   1:  PR[GP1:91,1] = PR[GP1:90,1] + 45.256;
   1:  PR[GP1:91,2] = PR[GP1:90,2] + 33.869;
   1:L PR[91] 10mm/sec CNT100;
   1:  PR[GP1:91,1] = PR[GP1:90,1] + 42.073;
   1:  PR[GP1:91,2] = PR[GP1:90,2] + 34.713;
   1:L PR[91] 10mm/sec CNT100;
   1:  PR[GP1:91,1] = PR[GP1:90,1] + 30.579;
   1:  PR[GP1:91,2] = PR[GP1:90,2] + 34.067;
   1:L PR[91] 10mm/sec CNT100;
   1:  PR[GP1:91,1] = PR[GP1:90,1] + 29.717;
   1:  PR[GP1:91,2] = PR[GP1:90,2] + 33.970;
   1:L PR[91] 10mm/sec CNT100;
   1:  PR[GP1:91,1] = PR[GP1:90,1] + 25.402;
   1:  PR[GP1:91,2] = PR[GP1:90,2] + 32.076;
   1:L PR[91] 10mm/sec CNT100;
   1:  PR[GP1:91,1] = PR[GP1:90,1] + 18.379;
   1:  PR[GP1:91,2] = PR[GP1:90,2] + 29.146;
   1:L PR[91] 10mm/sec CNT100;
   1:  PR[GP1:91,1] = PR[GP1:90,1] + 17.053;
   1:  PR[GP1:91,2] = PR[GP1:90,2] + 28.085;
   1:L PR[91] 10mm/sec CNT100;
   1:  PR[GP1:91,1] = PR[GP1:90,1] + 9.465;
   1:  PR[GP1:91,2] = PR[GP1:90,2] + 20.933;
   1:L PR[91] 10mm/sec CNT100;
   1:  PR[GP1:91,1] = PR[GP1:90,1] + 7.394;
   1:  PR[GP1:91,2] = PR[GP1:90,2] + 17.518;
   1:L PR[91] 10mm/sec CNT100;
   1:  PR[GP1:91,1] = PR[GP1:90,1] + 3.717;
   1:  PR[GP1:91,2] = PR[GP1:90,2] + 9.866;
   1:L PR[91] 10mm/sec CNT100;
   1:  PR[GP1:91,1] = PR[GP1:90,1] + -4.263;
   1:L PR[91] 10mm/sec CNT100;
   1:  PR[GP1:91,1] = PR[GP1:90,1] + -7.931;
   1:  PR[GP1:91,2] = PR[GP1:90,2] + 17.537;
   1:L PR[91] 10mm/sec CNT100;
   1:  PR[GP1:91,1] = PR[GP1:90,1] + -10.000;
   1:  PR[GP1:91,2] = PR[GP1:90,2] + 20.955;
   1:L PR[91] 10mm/sec CNT100;
   1:  PR[GP1:91,1] = PR[GP1:90,1] + -17.593;
   1:  PR[GP1:91,2] = PR[GP1:90,2] + 28.093;
   1:L PR[91] 10mm/sec CNT100;
   1:  PR[GP1:91,1] = PR[GP1:90,1] + -18.917;
   1:  PR[GP1:91,2] = PR[GP1:90,2] + 29.150;
   1:L PR[91] 10mm/sec CNT100;
   1:  PR[GP1:91,1] = PR[GP1:90,1] + -25.929;
   1:  PR[GP1:91,2] = PR[GP1:90,2] + 32.075;
   1:L PR[91] 10mm/sec CNT100;
   1:  PR[GP1:91,1] = PR[GP1:90,1] + -30.255;
   1:  PR[GP1:91,2] = PR[GP1:90,2] + 33.974;
   1:L PR[91] 10mm/sec CNT100;
   1:  PR[GP1:91,1] = PR[GP1:90,1] + -31.120;
   1:  PR[GP1:91,2] = PR[GP1:90,2] + 34.071;
   1:L PR[91] 10mm/sec CNT100;
   1:  PR[GP1:91,1] = PR[GP1:90,1] + -42.608;
   1:  PR[GP1:91,2] = PR[GP1:90,2] + 34.711;
   1:L PR[91] 10mm/sec CNT100;
   1:  PR[GP1:91,1] = PR[GP1:90,1] + -45.793;
   1:  PR[GP1:91,2] = PR[GP1:90,2] + 33.866;
   1:L PR[91] 10mm/sec CNT100;
   1:  PR[GP1:91,1] = PR[GP1:90,1] + -54.608;
   1:  PR[GP1:91,2] = PR[GP1:90,2] + 31.119;
   1:L PR[91] 10mm/sec CNT100;
   1:  PR[GP1:91,1] = PR[GP1:90,1] + -58.773;
   1:  PR[GP1:91,2] = PR[GP1:90,2] + 28.074;
   1:L PR[91] 10mm/sec CNT100;
   1:  PR[GP1:91,1] = PR[GP1:90,1] + -64.659;
   1:  PR[GP1:91,2] = PR[GP1:90,2] + 23.496;
   1:L PR[91] 10mm/sec CNT100;
   1:  PR[GP1:91,1] = PR[GP1:90,1] + -68.074;
   1:  PR[GP1:91,2] = PR[GP1:90,2] + 18.107;
   1:L PR[91] 10mm/sec CNT100;
   1:  PR[GP1:91,1] = PR[GP1:90,1] + -71.344;
   1:  PR[GP1:91,2] = PR[GP1:90,2] + 12.729;
   1:L PR[91] 10mm/sec CNT100;
   1:  PR[GP1:91,1] = PR[GP1:90,1] + -72.694;
   1:  PR[GP1:91,2] = PR[GP1:90,2] + 5.689;
   1:L PR[91] 10mm/sec CNT100;
   1:  PR[GP1:91,1] = PR[GP1:90,1] + -73.693;
   1:  PR[GP1:91,2] = PR[GP1:90,2] + 0.281;
   1:L PR[91] 10mm/sec CNT100;
   1:  PR[GP1:91,1] = PR[GP1:90,1] + -72.360;
   1:  PR[GP1:91,2] = PR[GP1:90,2] + -6.656;
   1:L PR[91] 10mm/sec CNT100;
   1:  PR[GP1:91,1] = PR[GP1:90,1] + -71.343;
   1:  PR[GP1:91,2] = PR[GP1:90,2] + -12.173;
   1:L PR[91] 10mm/sec CNT100;
   1:  PR[GP1:91,1] = PR[GP1:90,1] + -68.074;
   1:  PR[GP1:91,2] = PR[GP1:90,2] + -17.549;
   1:L PR[91] 10mm/sec CNT100;
   1:  PR[GP1:91,1] = PR[GP1:90,1] + -64.659;
   1:  PR[GP1:91,2] = PR[GP1:90,2] + -22.938;
   1:L PR[91] 10mm/sec CNT100;
   1:  PR[GP1:91,1] = PR[GP1:90,1] + -58.773;
   1:  PR[GP1:91,2] = PR[GP1:90,2] + -27.516;
   1:L PR[91] 10mm/sec CNT100;
   1:  PR[GP1:91,1] = PR[GP1:90,1] + -54.608;
   1:  PR[GP1:91,2] = PR[GP1:90,2] + -30.561;
   1:L PR[91] 10mm/sec CNT100;
   1:  PR[GP1:91,1] = PR[GP1:90,1] + -45.793;
   1:  PR[GP1:91,2] = PR[GP1:90,2] + -33.308;
   1:L PR[91] 10mm/sec CNT100;
   1:  PR[GP1:91,1] = PR[GP1:90,1] + -42.608;
   1:  PR[GP1:91,2] = PR[GP1:90,2] + -34.153;
   1:L PR[91] 10mm/sec CNT100;
   1:  PR[GP1:91,1] = PR[GP1:90,1] + -31.120;
   1:  PR[GP1:91,2] = PR[GP1:90,2] + -33.513;
   1:L PR[91] 10mm/sec CNT100;
   1:  PR[GP1:91,1] = PR[GP1:90,1] + -30.255;
   1:  PR[GP1:91,2] = PR[GP1:90,2] + -33.416;
   1:L PR[91] 10mm/sec CNT100;
   1:  PR[GP1:91,1] = PR[GP1:90,1] + -25.929;
   1:  PR[GP1:91,2] = PR[GP1:90,2] + -31.517;
   1:L PR[91] 10mm/sec CNT100;
   1:  PR[GP1:91,1] = PR[GP1:90,1] + -18.917;
   1:  PR[GP1:91,2] = PR[GP1:90,2] + -28.592;
   1:L PR[91] 10mm/sec CNT100;
   1:  PR[GP1:91,1] = PR[GP1:90,1] + -17.593;
   1:  PR[GP1:91,2] = PR[GP1:90,2] + -27.535;
   1:L PR[91] 10mm/sec CNT100;
   1:  PR[GP1:91,1] = PR[GP1:90,1] + -10.000;
   1:  PR[GP1:91,2] = PR[GP1:90,2] + -20.397;
   1:L PR[91] 10mm/sec CNT100;
   1:  PR[GP1:91,1] = PR[GP1:90,1] + -7.931;
   1:  PR[GP1:91,2] = PR[GP1:90,2] + -16.979;
   1:L PR[91] 10mm/sec CNT100;
   1:  PR[GP1:91,1] = PR[GP1:90,1] + -4.250;
   1:  PR[GP1:91,2] = PR[GP1:90,2] + -9.308;
   1:L PR[91] 10mm/sec CNT100;
   1:  PR[GP1:91,1] = PR[GP1:90,1] + 3.730;
   1:L PR[91] 10mm/sec CNT100;
   1:  PR[GP1:91,1] = PR[GP1:90,1] + 6.788;
   1:  PR[GP1:91,2] = PR[GP1:90,2] + -16.217;
   1:  PR[GP1:91,3] = PR[GP1:90,3] + 25.925;
   1:L PR[91] 10mm/sec CNT100;
   1:  PR[GP1:91,1] = PR[GP1:90,1] + 9.452;
   1:  PR[GP1:91,2] = PR[GP1:90,2] + -20.613;
   1:L PR[91] 10mm/sec CNT100;
   1:  PR[GP1:91,1] = PR[GP1:90,1] + 16.180;
   1:  PR[GP1:91,2] = PR[GP1:90,2] + -26.953;
   1:L PR[91] 10mm/sec CNT100;
   1:  PR[GP1:91,1] = PR[GP1:90,1] + 18.397;
   1:  PR[GP1:91,2] = PR[GP1:90,2] + -28.727;
   1:L PR[91] 10mm/sec CNT100;
   1:  PR[GP1:91,1] = PR[GP1:90,1] + 29.756;
   1:  PR[GP1:91,2] = PR[GP1:90,2] + -33.465;
   1:L PR[91] 10mm/sec CNT100;
   1:  PR[GP1:91,1] = PR[GP1:90,1] + 42.107;
   1:  PR[GP1:91,2] = PR[GP1:90,2] + -34.158;
   1:L PR[91] 10mm/sec CNT100;
   1:  PR[GP1:91,1] = PR[GP1:90,1] + 44.426;
   1:  PR[GP1:91,2] = PR[GP1:90,2] + -33.543;
   1:L PR[91] 10mm/sec CNT100;
   1:  PR[GP1:91,1] = PR[GP1:90,1] + 54.074;
   1:  PR[GP1:91,2] = PR[GP1:90,2] + -30.539;
   1:L PR[91] 10mm/sec CNT100;
   1:  PR[GP1:91,1] = PR[GP1:90,1] + 57.584;
   1:  PR[GP1:91,2] = PR[GP1:90,2] + -27.974;
   1:L PR[91] 10mm/sec CNT100;
   1:  PR[GP1:91,1] = PR[GP1:90,1] + 64.095;
   1:  PR[GP1:91,2] = PR[GP1:90,2] + -22.908;
   1:L PR[91] 10mm/sec CNT100;
   1:  PR[GP1:91,1] = PR[GP1:90,1] + 67.111;
   1:  PR[GP1:91,2] = PR[GP1:90,2] + -18.151;
   1:L PR[91] 10mm/sec CNT100;
   1:  PR[GP1:91,1] = PR[GP1:90,1] + 70.759;
   1:  PR[GP1:91,2] = PR[GP1:90,2] + -12.160;
   1:L PR[91] 10mm/sec CNT100;
   1:  PR[GP1:91,1] = PR[GP1:90,1] + 71.975;
   1:  PR[GP1:91,2] = PR[GP1:90,2] + -5.822;
   1:L PR[91] 10mm/sec CNT100;
   1:  PR[GP1:91,1] = PR[GP1:90,1] + 73.100;
   1:  PR[GP1:91,2] = PR[GP1:90,2] + 0.277;
   1:L PR[91] 10mm/sec CNT100;
   1:  PR[GP1:91,1] = PR[GP1:90,1] + 71.893;
   1:  PR[GP1:91,2] = PR[GP1:90,2] + 6.560;
   1:L PR[91] 10mm/sec CNT100;
   1:  PR[GP1:91,1] = PR[GP1:90,1] + 70.758;
   1:  PR[GP1:91,2] = PR[GP1:90,2] + 12.720;
   1:L PR[91] 10mm/sec CNT100;
   1:  PR[GP1:91,1] = PR[GP1:90,1] + 67.111;
   1:  PR[GP1:91,2] = PR[GP1:90,2] + 18.709;
   1:L PR[91] 10mm/sec CNT100;
   1:  PR[GP1:91,1] = PR[GP1:90,1] + 64.095;
   1:  PR[GP1:91,2] = PR[GP1:90,2] + 23.467;
   1:L PR[91] 10mm/sec CNT100;
   1:  PR[GP1:91,1] = PR[GP1:90,1] + 57.584;
   1:  PR[GP1:91,2] = PR[GP1:90,2] + 28.532;
   1:L PR[91] 10mm/sec CNT100;
   1:  PR[GP1:91,1] = PR[GP1:90,1] + 54.074;
   1:  PR[GP1:91,2] = PR[GP1:90,2] + 31.097;
   1:L PR[91] 10mm/sec CNT100;
   1:  PR[GP1:91,1] = PR[GP1:90,1] + 44.426;
   1:  PR[GP1:91,2] = PR[GP1:90,2] + 34.101;
   1:L PR[91] 10mm/sec CNT100;
   1:  PR[GP1:91,1] = PR[GP1:90,1] + 42.107;
   1:  PR[GP1:91,2] = PR[GP1:90,2] + 34.716;
   1:L PR[91] 10mm/sec CNT100;
   1:  PR[GP1:91,1] = PR[GP1:90,1] + 29.756;
   1:  PR[GP1:91,2] = PR[GP1:90,2] + 34.023;
   1:L PR[91] 10mm/sec CNT100;
   1:  PR[GP1:91,1] = PR[GP1:90,1] + 18.397;
   1:  PR[GP1:91,2] = PR[GP1:90,2] + 29.285;
   1:L PR[91] 10mm/sec CNT100;
   1:  PR[GP1:91,1] = PR[GP1:90,1] + 16.180;
   1:  PR[GP1:91,2] = PR[GP1:90,2] + 27.511;
   1:L PR[91] 10mm/sec CNT100;
   1:  PR[GP1:91,1] = PR[GP1:90,1] + 9.452;
   1:  PR[GP1:91,2] = PR[GP1:90,2] + 21.171;
   1:L PR[91] 10mm/sec CNT100;
   1:  PR[GP1:91,1] = PR[GP1:90,1] + 6.788;
   1:  PR[GP1:91,2] = PR[GP1:90,2] + 16.775;
   1:L PR[91] 10mm/sec CNT100;
   1:  PR[GP1:91,1] = PR[GP1:90,1] + 3.623;
   1:  PR[GP1:91,2] = PR[GP1:90,2] + 10.191;
   1:L PR[91] 10mm/sec CNT100;
   1:  PR[GP1:91,1] = PR[GP1:90,1] + -4.168;
   1:L PR[91] 10mm/sec CNT100;
   1:  PR[GP1:91,1] = PR[GP1:90,1] + -7.325;
   1:  PR[GP1:91,2] = PR[GP1:90,2] + 16.792;
   1:L PR[91] 10mm/sec CNT100;
   1:  PR[GP1:91,1] = PR[GP1:90,1] + -9.987;
   1:  PR[GP1:91,2] = PR[GP1:90,2] + 21.192;
   1:L PR[91] 10mm/sec CNT100;
   1:  PR[GP1:91,1] = PR[GP1:90,1] + -16.719;
   1:  PR[GP1:91,2] = PR[GP1:90,2] + 27.520;
   1:L PR[91] 10mm/sec CNT100;
   1:  PR[GP1:91,1] = PR[GP1:90,1] + -18.934;
   1:  PR[GP1:91,2] = PR[GP1:90,2] + 29.289;
   1:L PR[91] 10mm/sec CNT100;
   1:  PR[GP1:91,1] = PR[GP1:90,1] + -30.295;
   1:  PR[GP1:91,2] = PR[GP1:90,2] + 34.027;
   1:L PR[91] 10mm/sec CNT100;
   1:  PR[GP1:91,1] = PR[GP1:90,1] + -42.643;
   1:  PR[GP1:91,2] = PR[GP1:90,2] + 34.715;
   1:L PR[91] 10mm/sec CNT100;
   1:  PR[GP1:91,1] = PR[GP1:90,1] + -44.963;
   1:  PR[GP1:91,2] = PR[GP1:90,2] + 34.099;
   1:L PR[91] 10mm/sec CNT100;
   1:  PR[GP1:91,1] = PR[GP1:90,1] + -54.606;
   1:  PR[GP1:91,2] = PR[GP1:90,2] + 31.094;
   1:L PR[91] 10mm/sec CNT100;
   1:  PR[GP1:91,1] = PR[GP1:90,1] + -58.116;
   1:  PR[GP1:91,2] = PR[GP1:90,2] + 28.528;
   1:L PR[91] 10mm/sec CNT100;
   1:  PR[GP1:91,1] = PR[GP1:90,1] + -64.624;
   1:  PR[GP1:91,2] = PR[GP1:90,2] + 23.466;
   1:L PR[91] 10mm/sec CNT100;
   1:  PR[GP1:91,1] = PR[GP1:90,1] + -67.640;
   1:  PR[GP1:91,2] = PR[GP1:90,2] + 18.707;
   1:L PR[91] 10mm/sec CNT100;
   1:  PR[GP1:91,1] = PR[GP1:90,1] + -71.286;
   1:  PR[GP1:91,2] = PR[GP1:90,2] + 12.709;
   1:L PR[91] 10mm/sec CNT100;
   1:  PR[GP1:91,1] = PR[GP1:90,1] + -72.501;
   1:  PR[GP1:91,2] = PR[GP1:90,2] + 6.373;
   1:L PR[91] 10mm/sec CNT100;
   1:  PR[GP1:91,1] = PR[GP1:90,1] + -73.627;
   1:  PR[GP1:91,2] = PR[GP1:90,2] + 0.281;
   1:L PR[91] 10mm/sec CNT100;
   1:  PR[GP1:91,1] = PR[GP1:90,1] + -72.420;
   1:  PR[GP1:91,2] = PR[GP1:90,2] + -6.000;
   1:L PR[91] 10mm/sec CNT100;
   1:  PR[GP1:91,1] = PR[GP1:90,1] + -71.285;
   1:  PR[GP1:91,2] = PR[GP1:90,2] + -12.153;
   1:L PR[91] 10mm/sec CNT100;
   1:  PR[GP1:91,1] = PR[GP1:90,1] + -67.640;
   1:  PR[GP1:91,2] = PR[GP1:90,2] + -18.149;
   1:L PR[91] 10mm/sec CNT100;
   1:  PR[GP1:91,1] = PR[GP1:90,1] + -64.624;
   1:  PR[GP1:91,2] = PR[GP1:90,2] + -22.908;
   1:L PR[91] 10mm/sec CNT100;
   1:  PR[GP1:91,1] = PR[GP1:90,1] + -58.116;
   1:  PR[GP1:91,2] = PR[GP1:90,2] + -27.970;
   1:L PR[91] 10mm/sec CNT100;
   1:  PR[GP1:91,1] = PR[GP1:90,1] + -54.606;
   1:  PR[GP1:91,2] = PR[GP1:90,2] + -30.536;
   1:L PR[91] 10mm/sec CNT100;
   1:  PR[GP1:91,1] = PR[GP1:90,1] + -44.963;
   1:  PR[GP1:91,2] = PR[GP1:90,2] + -33.541;
   1:L PR[91] 10mm/sec CNT100;
   1:  PR[GP1:91,1] = PR[GP1:90,1] + -42.643;
   1:  PR[GP1:91,2] = PR[GP1:90,2] + -34.157;
   1:L PR[91] 10mm/sec CNT100;
   1:  PR[GP1:91,1] = PR[GP1:90,1] + -30.294;
   1:  PR[GP1:91,2] = PR[GP1:90,2] + -33.469;
   1:L PR[91] 10mm/sec CNT100;
   1:  PR[GP1:91,1] = PR[GP1:90,1] + -18.934;
   1:  PR[GP1:91,2] = PR[GP1:90,2] + -28.731;
   1:L PR[91] 10mm/sec CNT100;
   1:  PR[GP1:91,1] = PR[GP1:90,1] + -16.719;
   1:  PR[GP1:91,2] = PR[GP1:90,2] + -26.962;
   1:L PR[91] 10mm/sec CNT100;
   1:  PR[GP1:91,1] = PR[GP1:90,1] + -9.987;
   1:  PR[GP1:91,2] = PR[GP1:90,2] + -20.634;
   1:L PR[91] 10mm/sec CNT100;
   1:  PR[GP1:91,1] = PR[GP1:90,1] + -7.325;
   1:  PR[GP1:91,2] = PR[GP1:90,2] + -16.234;
   1:L PR[91] 10mm/sec CNT100;
   1:  PR[GP1:91,1] = PR[GP1:90,1] + -4.156;
   1:  PR[GP1:91,2] = PR[GP1:90,2] + -9.633;
   1:L PR[91] 10mm/sec CNT100;
   1:  PR[GP1:91,1] = PR[GP1:90,1] + 3.635;
   1:L PR[91] 10mm/sec CNT100;
   1:  PR[GP1:91,1] = PR[GP1:90,1] + 6.181;
   1:  PR[GP1:91,2] = PR[GP1:90,2] + -15.475;
   1:  PR[GP1:91,3] = PR[GP1:90,3] + 26.535;
   1:L PR[91] 10mm/sec CNT100;
   1:  PR[GP1:91,1] = PR[GP1:90,1] + 9.440;
   1:  PR[GP1:91,2] = PR[GP1:90,2] + -20.850;
   1:L PR[91] 10mm/sec CNT100;
   1:  PR[GP1:91,1] = PR[GP1:90,1] + 15.306;
   1:  PR[GP1:91,2] = PR[GP1:90,2] + -26.379;
   1:L PR[91] 10mm/sec CNT100;
   1:  PR[GP1:91,1] = PR[GP1:90,1] + 18.414;
   1:  PR[GP1:91,2] = PR[GP1:90,2] + -28.866;
   1:L PR[91] 10mm/sec CNT100;
   1:  PR[GP1:91,1] = PR[GP1:90,1] + 28.796;
   1:  PR[GP1:91,2] = PR[GP1:90,2] + -33.197;
   1:L PR[91] 10mm/sec CNT100;
   1:  PR[GP1:91,1] = PR[GP1:90,1] + 29.743;
   1:  PR[GP1:91,2] = PR[GP1:90,2] + -33.523;
   1:L PR[91] 10mm/sec CNT100;
   1:  PR[GP1:91,1] = PR[GP1:90,1] + 34.189;
   1:  PR[GP1:91,2] = PR[GP1:90,2] + -33.715;
   1:L PR[91] 10mm/sec CNT100;
   1:  PR[GP1:91,1] = PR[GP1:90,1] + 42.141;
   1:  PR[GP1:91,2] = PR[GP1:90,2] + -34.162;
   1:L PR[91] 10mm/sec CNT100;
   1:  PR[GP1:91,1] = PR[GP1:90,1] + 43.595;
   1:  PR[GP1:91,2] = PR[GP1:90,2] + -33.776;
   1:L PR[91] 10mm/sec CNT100;
   1:  PR[GP1:91,1] = PR[GP1:90,1] + 54.072;
   1:  PR[GP1:91,2] = PR[GP1:90,2] + -30.514;
   1:L PR[91] 10mm/sec CNT100;
   1:  PR[GP1:91,1] = PR[GP1:90,1] + 56.927;
   1:  PR[GP1:91,2] = PR[GP1:90,2] + -28.427;
   1:L PR[91] 10mm/sec CNT100;
   1:  PR[GP1:91,1] = PR[GP1:90,1] + 64.059;
   1:  PR[GP1:91,2] = PR[GP1:90,2] + -22.878;
   1:L PR[91] 10mm/sec CNT100;
   1:  PR[GP1:91,1] = PR[GP1:90,1] + 66.677;
   1:  PR[GP1:91,2] = PR[GP1:90,2] + -18.750;
   1:L PR[91] 10mm/sec CNT100;
   1:  PR[GP1:91,1] = PR[GP1:90,1] + 70.701;
   1:  PR[GP1:91,2] = PR[GP1:90,2] + -12.140;
   1:L PR[91] 10mm/sec CNT100;
   1:  PR[GP1:91,1] = PR[GP1:90,1] + 71.782;
   1:  PR[GP1:91,2] = PR[GP1:90,2] + -6.507;
   1:L PR[91] 10mm/sec CNT100;
   1:  PR[GP1:91,1] = PR[GP1:90,1] + 73.034;
   1:  PR[GP1:91,2] = PR[GP1:90,2] + 0.277;
   1:L PR[91] 10mm/sec CNT100;
   1:  PR[GP1:91,1] = PR[GP1:90,1] + 71.953;
   1:  PR[GP1:91,2] = PR[GP1:90,2] + 5.904;
   1:L PR[91] 10mm/sec CNT100;
   1:  PR[GP1:91,1] = PR[GP1:90,1] + 70.700;
   1:  PR[GP1:91,2] = PR[GP1:90,2] + 12.700;
   1:L PR[91] 10mm/sec CNT100;
   1:  PR[GP1:91,1] = PR[GP1:90,1] + 66.677;
   1:  PR[GP1:91,2] = PR[GP1:90,2] + 19.308;
   1:L PR[91] 10mm/sec CNT100;
   1:  PR[GP1:91,1] = PR[GP1:90,1] + 64.059;
   1:  PR[GP1:91,2] = PR[GP1:90,2] + 23.436;
   1:L PR[91] 10mm/sec CNT100;
   1:  PR[GP1:91,1] = PR[GP1:90,1] + 56.927;
   1:  PR[GP1:91,2] = PR[GP1:90,2] + 28.985;
   1:L PR[91] 10mm/sec CNT100;
   1:  PR[GP1:91,1] = PR[GP1:90,1] + 54.072;
   1:  PR[GP1:91,2] = PR[GP1:90,2] + 31.072;
   1:L PR[91] 10mm/sec CNT100;
   1:  PR[GP1:91,1] = PR[GP1:90,1] + 43.595;
   1:  PR[GP1:91,2] = PR[GP1:90,2] + 34.334;
   1:L PR[91] 10mm/sec CNT100;
   1:  PR[GP1:91,1] = PR[GP1:90,1] + 42.141;
   1:  PR[GP1:91,2] = PR[GP1:90,2] + 34.720;
   1:L PR[91] 10mm/sec CNT100;
   1:  PR[GP1:91,1] = PR[GP1:90,1] + 34.189;
   1:  PR[GP1:91,2] = PR[GP1:90,2] + 34.273;
   1:L PR[91] 10mm/sec CNT100;
   1:  PR[GP1:91,1] = PR[GP1:90,1] + 29.743;
   1:  PR[GP1:91,2] = PR[GP1:90,2] + 34.081;
   1:L PR[91] 10mm/sec CNT100;
   1:  PR[GP1:91,1] = PR[GP1:90,1] + 28.796;
   1:  PR[GP1:91,2] = PR[GP1:90,2] + 33.755;
   1:L PR[91] 10mm/sec CNT100;
   1:  PR[GP1:91,1] = PR[GP1:90,1] + 18.414;
   1:  PR[GP1:91,2] = PR[GP1:90,2] + 29.424;
   1:L PR[91] 10mm/sec CNT100;
   1:  PR[GP1:91,1] = PR[GP1:90,1] + 15.306;
   1:  PR[GP1:91,2] = PR[GP1:90,2] + 26.937;
   1:L PR[91] 10mm/sec CNT100;
   1:  PR[GP1:91,1] = PR[GP1:90,1] + 9.440;
   1:  PR[GP1:91,2] = PR[GP1:90,2] + 21.408;
   1:L PR[91] 10mm/sec CNT100;
   1:  PR[GP1:91,1] = PR[GP1:90,1] + 6.181;
   1:  PR[GP1:91,2] = PR[GP1:90,2] + 16.033;
   1:L PR[91] 10mm/sec CNT100;
   1:  PR[GP1:91,1] = PR[GP1:90,1] + 3.530;
   1:  PR[GP1:91,2] = PR[GP1:90,2] + 10.516;
   1:L PR[91] 10mm/sec CNT100;
   1:  PR[GP1:91,1] = PR[GP1:90,1] + -4.073;
   1:L PR[91] 10mm/sec CNT100;
   1:  PR[GP1:91,1] = PR[GP1:90,1] + -6.718;
   1:  PR[GP1:91,2] = PR[GP1:90,2] + 16.047;
   1:L PR[91] 10mm/sec CNT100;
   1:  PR[GP1:91,1] = PR[GP1:90,1] + -9.974;
   1:  PR[GP1:91,2] = PR[GP1:90,2] + 21.428;
   1:L PR[91] 10mm/sec CNT100;
   1:  PR[GP1:91,1] = PR[GP1:90,1] + -15.844;
   1:  PR[GP1:91,2] = PR[GP1:90,2] + 26.947;
   1:L PR[91] 10mm/sec CNT100;
   1:  PR[GP1:91,1] = PR[GP1:90,1] + -18.951;
   1:  PR[GP1:91,2] = PR[GP1:90,2] + 29.428;
   1:L PR[91] 10mm/sec CNT100;
   1:  PR[GP1:91,1] = PR[GP1:90,1] + -29.337;
   1:  PR[GP1:91,2] = PR[GP1:90,2] + 33.760;
   1:L PR[91] 10mm/sec CNT100;
   1:  PR[GP1:91,1] = PR[GP1:90,1] + -30.281;
   1:  PR[GP1:91,2] = PR[GP1:90,2] + 34.084;
   1:L PR[91] 10mm/sec CNT100;
   1:  PR[GP1:91,1] = PR[GP1:90,1] + -34.715;
   1:  PR[GP1:91,2] = PR[GP1:90,2] + 34.274;
   1:L PR[91] 10mm/sec CNT100;
   1:  PR[GP1:91,1] = PR[GP1:90,1] + -42.677;
   1:  PR[GP1:91,2] = PR[GP1:90,2] + 34.718;
   1:L PR[91] 10mm/sec CNT100;
   1:  PR[GP1:91,1] = PR[GP1:90,1] + -44.133;
   1:  PR[GP1:91,2] = PR[GP1:90,2] + 34.332;
   1:L PR[91] 10mm/sec CNT100;
   1:  PR[GP1:91,1] = PR[GP1:90,1] + -54.604;
   1:  PR[GP1:91,2] = PR[GP1:90,2] + 31.069;
   1:L PR[91] 10mm/sec CNT100;
   1:  PR[GP1:91,1] = PR[GP1:90,1] + -57.459;
   1:  PR[GP1:91,2] = PR[GP1:90,2] + 28.982;
   1:L PR[91] 10mm/sec CNT100;
   1:  PR[GP1:91,1] = PR[GP1:90,1] + -64.588;
   1:  PR[GP1:91,2] = PR[GP1:90,2] + 23.436;
   1:L PR[91] 10mm/sec CNT100;
   1:  PR[GP1:91,1] = PR[GP1:90,1] + -67.205;
   1:  PR[GP1:91,2] = PR[GP1:90,2] + 19.307;
   1:L PR[91] 10mm/sec CNT100;
   1:  PR[GP1:91,1] = PR[GP1:90,1] + -71.228;
   1:  PR[GP1:91,2] = PR[GP1:90,2] + 12.690;
   1:L PR[91] 10mm/sec CNT100;
   1:  PR[GP1:91,1] = PR[GP1:90,1] + -72.309;
   1:  PR[GP1:91,2] = PR[GP1:90,2] + 7.058;
   1:L PR[91] 10mm/sec CNT100;
   1:  PR[GP1:91,1] = PR[GP1:90,1] + -73.560;
   1:  PR[GP1:91,2] = PR[GP1:90,2] + 0.281;
   1:L PR[91] 10mm/sec CNT100;
   1:  PR[GP1:91,1] = PR[GP1:90,1] + -72.479;
   1:  PR[GP1:91,2] = PR[GP1:90,2] + -5.344;
   1:L PR[91] 10mm/sec CNT100;
   1:  PR[GP1:91,1] = PR[GP1:90,1] + -71.227;
   1:  PR[GP1:91,2] = PR[GP1:90,2] + -12.133;
   1:L PR[91] 10mm/sec CNT100;
   1:  PR[GP1:91,1] = PR[GP1:90,1] + -67.205;
   1:  PR[GP1:91,2] = PR[GP1:90,2] + -18.749;
   1:L PR[91] 10mm/sec CNT100;
   1:  PR[GP1:91,1] = PR[GP1:90,1] + -64.588;
   1:  PR[GP1:91,2] = PR[GP1:90,2] + -22.878;
   1:L PR[91] 10mm/sec CNT100;
   1:  PR[GP1:91,1] = PR[GP1:90,1] + -57.459;
   1:  PR[GP1:91,2] = PR[GP1:90,2] + -28.424;
   1:L PR[91] 10mm/sec CNT100;
   1:  PR[GP1:91,1] = PR[GP1:90,1] + -54.604;
   1:  PR[GP1:91,2] = PR[GP1:90,2] + -30.511;
   1:L PR[91] 10mm/sec CNT100;
   1:  PR[GP1:91,1] = PR[GP1:90,1] + -44.133;
   1:  PR[GP1:91,2] = PR[GP1:90,2] + -33.774;
   1:L PR[91] 10mm/sec CNT100;
   1:  PR[GP1:91,1] = PR[GP1:90,1] + -42.677;
   1:  PR[GP1:91,2] = PR[GP1:90,2] + -34.160;
   1:L PR[91] 10mm/sec CNT100;
   1:  PR[GP1:91,1] = PR[GP1:90,1] + -34.715;
   1:  PR[GP1:91,2] = PR[GP1:90,2] + -33.716;
   1:L PR[91] 10mm/sec CNT100;
   1:  PR[GP1:91,1] = PR[GP1:90,1] + -30.281;
   1:  PR[GP1:91,2] = PR[GP1:90,2] + -33.526;
   1:L PR[91] 10mm/sec CNT100;
   1:  PR[GP1:91,1] = PR[GP1:90,1] + -29.337;
   1:  PR[GP1:91,2] = PR[GP1:90,2] + -33.202;
   1:L PR[91] 10mm/sec CNT100;
   1:  PR[GP1:91,1] = PR[GP1:90,1] + -18.951;
   1:  PR[GP1:91,2] = PR[GP1:90,2] + -28.870;
   1:L PR[91] 10mm/sec CNT100;
   1:  PR[GP1:91,1] = PR[GP1:90,1] + -15.844;
   1:  PR[GP1:91,2] = PR[GP1:90,2] + -26.389;
   1:L PR[91] 10mm/sec CNT100;
   1:  PR[GP1:91,1] = PR[GP1:90,1] + -9.974;
   1:  PR[GP1:91,2] = PR[GP1:90,2] + -20.870;
   1:L PR[91] 10mm/sec CNT100;
   1:  PR[GP1:91,1] = PR[GP1:90,1] + -6.718;
   1:  PR[GP1:91,2] = PR[GP1:90,2] + -15.489;
   1:L PR[91] 10mm/sec CNT100;
   1:  PR[GP1:91,1] = PR[GP1:90,1] + -4.063;
   1:  PR[GP1:91,2] = PR[GP1:90,2] + -9.958;
   1:L PR[91] 10mm/sec CNT100;
   1:  PR[GP1:91,1] = PR[GP1:90,1] + 3.539;
   1:L PR[91] 10mm/sec CNT100;
   1:  PR[GP1:91,1] = PR[GP1:90,1] + 5.574;
   1:  PR[GP1:91,2] = PR[GP1:90,2] + -14.732;
   1:  PR[GP1:91,3] = PR[GP1:90,3] + 27.145;
   1:L PR[91] 10mm/sec CNT100;
   1:  PR[GP1:91,1] = PR[GP1:90,1] + 9.427;
   1:  PR[GP1:91,2] = PR[GP1:90,2] + -21.088;
   1:L PR[91] 10mm/sec CNT100;
   1:  PR[GP1:91,1] = PR[GP1:90,1] + 14.433;
   1:  PR[GP1:91,2] = PR[GP1:90,2] + -25.806;
   1:L PR[91] 10mm/sec CNT100;
   1:  PR[GP1:91,1] = PR[GP1:90,1] + 18.432;
   1:  PR[GP1:91,2] = PR[GP1:90,2] + -29.005;
   1:L PR[91] 10mm/sec CNT100;
   1:  PR[GP1:91,1] = PR[GP1:90,1] + 27.770;
   1:  PR[GP1:91,2] = PR[GP1:90,2] + -32.901;
   1:L PR[91] 10mm/sec CNT100;
   1:  PR[GP1:91,1] = PR[GP1:90,1] + 29.753;
   1:  PR[GP1:91,2] = PR[GP1:90,2] + -33.583;
   1:L PR[91] 10mm/sec CNT100;
   1:  PR[GP1:91,1] = PR[GP1:90,1] + 38.683;
   1:  PR[GP1:91,2] = PR[GP1:90,2] + -33.969;
   1:L PR[91] 10mm/sec CNT100;
   1:  PR[GP1:91,1] = PR[GP1:90,1] + 42.175;
   1:  PR[GP1:91,2] = PR[GP1:90,2] + -34.165;
   1:L PR[91] 10mm/sec CNT100;
   1:  PR[GP1:91,1] = PR[GP1:90,1] + 42.765;
   1:  PR[GP1:91,2] = PR[GP1:90,2] + -34.009;
   1:L PR[91] 10mm/sec CNT100;
   1:  PR[GP1:91,1] = PR[GP1:90,1] + 54.069;
   1:  PR[GP1:91,2] = PR[GP1:90,2] + -30.489;
   1:L PR[91] 10mm/sec CNT100;
   1:  PR[GP1:91,1] = PR[GP1:90,1] + 56.269;
   1:  PR[GP1:91,2] = PR[GP1:90,2] + -28.881;
   1:L PR[91] 10mm/sec CNT100;
   1:  PR[GP1:91,1] = PR[GP1:90,1] + 64.024;
   1:  PR[GP1:91,2] = PR[GP1:90,2] + -22.848;
   1:L PR[91] 10mm/sec CNT100;
   1:  PR[GP1:91,1] = PR[GP1:90,1] + 66.242;
   1:  PR[GP1:91,2] = PR[GP1:90,2] + -19.350;
   1:L PR[91] 10mm/sec CNT100;
   1:  PR[GP1:91,1] = PR[GP1:90,1] + 70.643;
   1:  PR[GP1:91,2] = PR[GP1:90,2] + -12.121;
   1:L PR[91] 10mm/sec CNT100;
   1:  PR[GP1:91,1] = PR[GP1:90,1] + 71.589;
   1:  PR[GP1:91,2] = PR[GP1:90,2] + -7.192;
   1:L PR[91] 10mm/sec CNT100;
   1:  PR[GP1:91,1] = PR[GP1:90,1] + 72.967;
   1:  PR[GP1:91,2] = PR[GP1:90,2] + 0.277;
   1:L PR[91] 10mm/sec CNT100;
   1:  PR[GP1:91,1] = PR[GP1:90,1] + 72.013;
   1:  PR[GP1:91,2] = PR[GP1:90,2] + 5.248;
   1:L PR[91] 10mm/sec CNT100;
   1:  PR[GP1:91,1] = PR[GP1:90,1] + 70.642;
   1:  PR[GP1:91,2] = PR[GP1:90,2] + 12.681;
   1:L PR[91] 10mm/sec CNT100;
   1:  PR[GP1:91,1] = PR[GP1:90,1] + 66.242;
   1:  PR[GP1:91,2] = PR[GP1:90,2] + 19.908;
   1:L PR[91] 10mm/sec CNT100;
   1:  PR[GP1:91,1] = PR[GP1:90,1] + 64.024;
   1:  PR[GP1:91,2] = PR[GP1:90,2] + 23.406;
   1:L PR[91] 10mm/sec CNT100;
   1:  PR[GP1:91,1] = PR[GP1:90,1] + 56.269;
   1:  PR[GP1:91,2] = PR[GP1:90,2] + 29.439;
   1:L PR[91] 10mm/sec CNT100;
   1:  PR[GP1:91,1] = PR[GP1:90,1] + 54.069;
   1:  PR[GP1:91,2] = PR[GP1:90,2] + 31.047;
   1:L PR[91] 10mm/sec CNT100;
   1:  PR[GP1:91,1] = PR[GP1:90,1] + 42.765;
   1:  PR[GP1:91,2] = PR[GP1:90,2] + 34.567;
   1:L PR[91] 10mm/sec CNT100;
   1:  PR[GP1:91,1] = PR[GP1:90,1] + 42.175;
   1:  PR[GP1:91,2] = PR[GP1:90,2] + 34.724;
   1:L PR[91] 10mm/sec CNT100;
   1:  PR[GP1:91,1] = PR[GP1:90,1] + 38.683;
   1:  PR[GP1:91,2] = PR[GP1:90,2] + 34.527;
   1:L PR[91] 10mm/sec CNT100;
   1:  PR[GP1:91,1] = PR[GP1:90,1] + 29.753;
   1:  PR[GP1:91,2] = PR[GP1:90,2] + 34.141;
   1:L PR[91] 10mm/sec CNT100;
   1:  PR[GP1:91,1] = PR[GP1:90,1] + 27.770;
   1:  PR[GP1:91,2] = PR[GP1:90,2] + 33.459;
   1:L PR[91] 10mm/sec CNT100;
   1:  PR[GP1:91,1] = PR[GP1:90,1] + 18.432;
   1:  PR[GP1:91,2] = PR[GP1:90,2] + 29.563;
   1:L PR[91] 10mm/sec CNT100;
   1:  PR[GP1:91,1] = PR[GP1:90,1] + 14.433;
   1:  PR[GP1:91,2] = PR[GP1:90,2] + 26.364;
   1:L PR[91] 10mm/sec CNT100;
   1:  PR[GP1:91,1] = PR[GP1:90,1] + 9.427;
   1:  PR[GP1:91,2] = PR[GP1:90,2] + 21.646;
   1:L PR[91] 10mm/sec CNT100;
   1:  PR[GP1:91,1] = PR[GP1:90,1] + 5.575;
   1:  PR[GP1:91,2] = PR[GP1:90,2] + 15.291;
   1:L PR[91] 10mm/sec CNT100;
   1:  PR[GP1:91,1] = PR[GP1:90,1] + 3.436;
   1:  PR[GP1:91,2] = PR[GP1:90,2] + 10.841;
   1:L PR[91] 10mm/sec CNT100;
   1:  PR[GP1:91,1] = PR[GP1:90,1] + -3.977;
   1:L PR[91] 10mm/sec CNT100;
   1:  PR[GP1:91,1] = PR[GP1:90,1] + -6.111;
   1:  PR[GP1:91,2] = PR[GP1:90,2] + 15.302;
   1:L PR[91] 10mm/sec CNT100;
   1:  PR[GP1:91,1] = PR[GP1:90,1] + -9.961;
   1:  PR[GP1:91,2] = PR[GP1:90,2] + 21.665;
   1:L PR[91] 10mm/sec CNT100;
   1:  PR[GP1:91,1] = PR[GP1:90,1] + -14.970;
   1:  PR[GP1:91,2] = PR[GP1:90,2] + 26.374;
   1:L PR[91] 10mm/sec CNT100;
   1:  PR[GP1:91,1] = PR[GP1:90,1] + -18.969;
   1:  PR[GP1:91,2] = PR[GP1:90,2] + 29.567;
   1:L PR[91] 10mm/sec CNT100;
   1:  PR[GP1:91,1] = PR[GP1:90,1] + -28.311;
   1:  PR[GP1:91,2] = PR[GP1:90,2] + 33.463;
   1:L PR[91] 10mm/sec CNT100;
   1:  PR[GP1:91,1] = PR[GP1:90,1] + -30.291;
   1:  PR[GP1:91,2] = PR[GP1:90,2] + 34.144;
   1:L PR[91] 10mm/sec CNT100;
   1:  PR[GP1:91,1] = PR[GP1:90,1] + -39.209;
   1:  PR[GP1:91,2] = PR[GP1:90,2] + 34.527;
   1:L PR[91] 10mm/sec CNT100;
   1:  PR[GP1:91,1] = PR[GP1:90,1] + -42.711;
   1:  PR[GP1:91,2] = PR[GP1:90,2] + 34.722;
   1:L PR[91] 10mm/sec CNT100;
   1:  PR[GP1:91,1] = PR[GP1:90,1] + -43.303;
   1:  PR[GP1:91,2] = PR[GP1:90,2] + 34.565;
   1:L PR[91] 10mm/sec CNT100;
   1:  PR[GP1:91,1] = PR[GP1:90,1] + -54.602;
   1:  PR[GP1:91,2] = PR[GP1:90,2] + 31.043;
   1:L PR[91] 10mm/sec CNT100;
   1:  PR[GP1:91,1] = PR[GP1:90,1] + -56.802;
   1:  PR[GP1:91,2] = PR[GP1:90,2] + 29.435;
   1:L PR[91] 10mm/sec CNT100;
   1:  PR[GP1:91,1] = PR[GP1:90,1] + -64.553;
   1:  PR[GP1:91,2] = PR[GP1:90,2] + 23.406;
   1:L PR[91] 10mm/sec CNT100;
   1:  PR[GP1:91,1] = PR[GP1:90,1] + -66.771;
   1:  PR[GP1:91,2] = PR[GP1:90,2] + 19.906;
   1:L PR[91] 10mm/sec CNT100;
   1:  PR[GP1:91,1] = PR[GP1:90,1] + -71.170;
   1:  PR[GP1:91,2] = PR[GP1:90,2] + 12.670;
   1:L PR[91] 10mm/sec CNT100;
   1:  PR[GP1:91,1] = PR[GP1:90,1] + -72.116;
   1:  PR[GP1:91,2] = PR[GP1:90,2] + 7.742;
   1:L PR[91] 10mm/sec CNT100;
   1:  PR[GP1:91,1] = PR[GP1:90,1] + -73.494;
   1:  PR[GP1:91,2] = PR[GP1:90,2] + 0.281;
   1:L PR[91] 10mm/sec CNT100;
   1:  PR[GP1:91,1] = PR[GP1:90,1] + -72.539;
   1:  PR[GP1:91,2] = PR[GP1:90,2] + -4.688;
   1:L PR[91] 10mm/sec CNT100;
   1:  PR[GP1:91,1] = PR[GP1:90,1] + -71.169;
   1:  PR[GP1:91,2] = PR[GP1:90,2] + -12.114;
   1:L PR[91] 10mm/sec CNT100;
   1:  PR[GP1:91,1] = PR[GP1:90,1] + -66.771;
   1:  PR[GP1:91,2] = PR[GP1:90,2] + -19.348;
   1:L PR[91] 10mm/sec CNT100;
   1:  PR[GP1:91,1] = PR[GP1:90,1] + -64.553;
   1:  PR[GP1:91,2] = PR[GP1:90,2] + -22.848;
   1:L PR[91] 10mm/sec CNT100;
   1:  PR[GP1:91,1] = PR[GP1:90,1] + -56.802;
   1:  PR[GP1:91,2] = PR[GP1:90,2] + -28.877;
   1:L PR[91] 10mm/sec CNT100;
   1:  PR[GP1:91,1] = PR[GP1:90,1] + -54.602;
   1:  PR[GP1:91,2] = PR[GP1:90,2] + -30.485;
   1:L PR[91] 10mm/sec CNT100;
   1:  PR[GP1:91,1] = PR[GP1:90,1] + -43.303;
   1:  PR[GP1:91,2] = PR[GP1:90,2] + -34.007;
   1:L PR[91] 10mm/sec CNT100;
   1:  PR[GP1:91,1] = PR[GP1:90,1] + -42.711;
   1:  PR[GP1:91,2] = PR[GP1:90,2] + -34.164;
   1:L PR[91] 10mm/sec CNT100;
   1:  PR[GP1:91,1] = PR[GP1:90,1] + -39.209;
   1:  PR[GP1:91,2] = PR[GP1:90,2] + -33.969;
   1:L PR[91] 10mm/sec CNT100;
   1:  PR[GP1:91,1] = PR[GP1:90,1] + -30.291;
   1:  PR[GP1:91,2] = PR[GP1:90,2] + -33.586;
   1:L PR[91] 10mm/sec CNT100;
   1:  PR[GP1:91,1] = PR[GP1:90,1] + -28.311;
   1:  PR[GP1:91,2] = PR[GP1:90,2] + -32.905;
   1:L PR[91] 10mm/sec CNT100;
   1:  PR[GP1:91,1] = PR[GP1:90,1] + -18.969;
   1:  PR[GP1:91,2] = PR[GP1:90,2] + -29.009;
   1:L PR[91] 10mm/sec CNT100;
   1:  PR[GP1:91,1] = PR[GP1:90,1] + -14.970;
   1:  PR[GP1:91,2] = PR[GP1:90,2] + -25.816;
   1:L PR[91] 10mm/sec CNT100;
   1:  PR[GP1:91,1] = PR[GP1:90,1] + -9.961;
   1:  PR[GP1:91,2] = PR[GP1:90,2] + -21.107;
   1:L PR[91] 10mm/sec CNT100;
   1:  PR[GP1:91,1] = PR[GP1:90,1] + -6.111;
   1:  PR[GP1:91,2] = PR[GP1:90,2] + -14.744;
   1:L PR[91] 10mm/sec CNT100;
   1:  PR[GP1:91,1] = PR[GP1:90,1] + -3.969;
   1:  PR[GP1:91,2] = PR[GP1:90,2] + -10.283;
   1:L PR[91] 10mm/sec CNT100;
   1:  PR[GP1:91,1] = PR[GP1:90,1] + 3.444;
   1:L PR[91] 10mm/sec CNT100;
   1:  PR[GP1:91,1] = PR[GP1:90,1] + 4.968;
   1:  PR[GP1:91,2] = PR[GP1:90,2] + -13.990;
   1:  PR[GP1:91,3] = PR[GP1:90,3] + 27.755;
   1:L PR[91] 10mm/sec CNT100;
   1:  PR[GP1:91,1] = PR[GP1:90,1] + 9.415;
   1:  PR[GP1:91,2] = PR[GP1:90,2] + -21.326;
   1:L PR[91] 10mm/sec CNT100;
   1:  PR[GP1:91,1] = PR[GP1:90,1] + 13.559;
   1:  PR[GP1:91,2] = PR[GP1:90,2] + -25.232;
   1:L PR[91] 10mm/sec CNT100;
   1:  PR[GP1:91,1] = PR[GP1:90,1] + 18.450;
   1:  PR[GP1:91,2] = PR[GP1:90,2] + -29.145;
   1:L PR[91] 10mm/sec CNT100;
   1:  PR[GP1:91,1] = PR[GP1:90,1] + 26.744;
   1:  PR[GP1:91,2] = PR[GP1:90,2] + -32.605;
   1:L PR[91] 10mm/sec CNT100;
   1:  PR[GP1:91,1] = PR[GP1:90,1] + 29.763;
   1:  PR[GP1:91,2] = PR[GP1:90,2] + -33.643;
   1:L PR[91] 10mm/sec CNT100;
   1:  PR[GP1:91,1] = PR[GP1:90,1] + 42.071;
   1:  PR[GP1:91,2] = PR[GP1:90,2] + -34.176;
   1:L PR[91] 10mm/sec CNT100;
   1:  PR[GP1:91,1] = PR[GP1:90,1] + 42.167;
   1:  PR[GP1:91,2] = PR[GP1:90,2] + -34.175;
   1:L PR[91] 10mm/sec CNT100;
   1:  PR[GP1:91,1] = PR[GP1:90,1] + 54.067;
   1:  PR[GP1:91,2] = PR[GP1:90,2] + -30.464;
   1:L PR[91] 10mm/sec CNT100;
   1:  PR[GP1:91,1] = PR[GP1:90,1] + 55.612;
   1:  PR[GP1:91,2] = PR[GP1:90,2] + -29.335;
   1:L PR[91] 10mm/sec CNT100;
   1:  PR[GP1:91,1] = PR[GP1:90,1] + 63.989;
   1:  PR[GP1:91,2] = PR[GP1:90,2] + -22.818;
   1:L PR[91] 10mm/sec CNT100;
   1:  PR[GP1:91,1] = PR[GP1:90,1] + 65.807;
   1:  PR[GP1:91,2] = PR[GP1:90,2] + -19.950;
   1:L PR[91] 10mm/sec CNT100;
   1:  PR[GP1:91,1] = PR[GP1:90,1] + 70.586;
   1:  PR[GP1:91,2] = PR[GP1:90,2] + -12.102;
   1:L PR[91] 10mm/sec CNT100;
   1:  PR[GP1:91,1] = PR[GP1:90,1] + 71.396;
   1:  PR[GP1:91,2] = PR[GP1:90,2] + -7.877;
   1:L PR[91] 10mm/sec CNT100;
   1:  PR[GP1:91,1] = PR[GP1:90,1] + 72.901;
   1:  PR[GP1:91,2] = PR[GP1:90,2] + 0.277;
   1:L PR[91] 10mm/sec CNT100;
   1:  PR[GP1:91,1] = PR[GP1:90,1] + 72.072;
   1:  PR[GP1:91,2] = PR[GP1:90,2] + 4.591;
   1:L PR[91] 10mm/sec CNT100;
   1:  PR[GP1:91,1] = PR[GP1:90,1] + 70.584;
   1:  PR[GP1:91,2] = PR[GP1:90,2] + 12.662;
   1:L PR[91] 10mm/sec CNT100;
   1:  PR[GP1:91,1] = PR[GP1:90,1] + 65.807;
   1:  PR[GP1:91,2] = PR[GP1:90,2] + 20.508;
   1:L PR[91] 10mm/sec CNT100;
   1:  PR[GP1:91,1] = PR[GP1:90,1] + 63.989;
   1:  PR[GP1:91,2] = PR[GP1:90,2] + 23.376;
   1:L PR[91] 10mm/sec CNT100;
   1:  PR[GP1:91,1] = PR[GP1:90,1] + 55.612;
   1:  PR[GP1:91,2] = PR[GP1:90,2] + 29.893;
   1:L PR[91] 10mm/sec CNT100;
   1:  PR[GP1:91,1] = PR[GP1:90,1] + 54.067;
   1:  PR[GP1:91,2] = PR[GP1:90,2] + 31.022;
   1:L PR[91] 10mm/sec CNT100;
   1:  PR[GP1:91,1] = PR[GP1:90,1] + 42.166;
   1:  PR[GP1:91,2] = PR[GP1:90,2] + 34.733;
   1:L PR[91] 10mm/sec CNT100;
   1:  PR[GP1:91,1] = PR[GP1:90,1] + 42.071;
   1:  PR[GP1:91,2] = PR[GP1:90,2] + 34.734;
   1:L PR[91] 10mm/sec CNT100;
   1:  PR[GP1:91,1] = PR[GP1:90,1] + 29.763;
   1:  PR[GP1:91,2] = PR[GP1:90,2] + 34.201;
   1:L PR[91] 10mm/sec CNT100;
   1:  PR[GP1:91,1] = PR[GP1:90,1] + 26.744;
   1:  PR[GP1:91,2] = PR[GP1:90,2] + 33.163;
   1:L PR[91] 10mm/sec CNT100;
   1:  PR[GP1:91,1] = PR[GP1:90,1] + 18.450;
   1:  PR[GP1:91,2] = PR[GP1:90,2] + 29.703;
   1:L PR[91] 10mm/sec CNT100;
   1:  PR[GP1:91,1] = PR[GP1:90,1] + 13.559;
   1:  PR[GP1:91,2] = PR[GP1:90,2] + 25.790;
   1:L PR[91] 10mm/sec CNT100;
   1:  PR[GP1:91,1] = PR[GP1:90,1] + 9.415;
   1:  PR[GP1:91,2] = PR[GP1:90,2] + 21.884;
   1:L PR[91] 10mm/sec CNT100;
   1:  PR[GP1:91,1] = PR[GP1:90,1] + 4.968;
   1:  PR[GP1:91,2] = PR[GP1:90,2] + 14.549;
   1:L PR[91] 10mm/sec CNT100;
   1:  PR[GP1:91,1] = PR[GP1:90,1] + 3.342;
   1:  PR[GP1:91,2] = PR[GP1:90,2] + 11.166;
   1:L PR[91] 10mm/sec CNT100;
   1:  PR[GP1:91,1] = PR[GP1:90,1] + -3.882;
   1:L PR[91] 10mm/sec CNT100;
   1:  PR[GP1:91,1] = PR[GP1:90,1] + -5.504;
   1:  PR[GP1:91,2] = PR[GP1:90,2] + 14.557;
   1:L PR[91] 10mm/sec CNT100;
   1:  PR[GP1:91,1] = PR[GP1:90,1] + -9.948;
   1:  PR[GP1:91,2] = PR[GP1:90,2] + 21.902;
   1:L PR[91] 10mm/sec CNT100;
   1:  PR[GP1:91,1] = PR[GP1:90,1] + -14.096;
   1:  PR[GP1:91,2] = PR[GP1:90,2] + 25.801;
   1:L PR[91] 10mm/sec CNT100;
   1:  PR[GP1:91,1] = PR[GP1:90,1] + -18.986;
   1:  PR[GP1:91,2] = PR[GP1:90,2] + 29.706;
   1:L PR[91] 10mm/sec CNT100;
   1:  PR[GP1:91,1] = PR[GP1:90,1] + -27.284;
   1:  PR[GP1:91,2] = PR[GP1:90,2] + 33.167;
   1:L PR[91] 10mm/sec CNT100;
   1:  PR[GP1:91,1] = PR[GP1:90,1] + -30.300;
   1:  PR[GP1:91,2] = PR[GP1:90,2] + 34.204;
   1:L PR[91] 10mm/sec CNT100;
   1:  PR[GP1:91,1] = PR[GP1:90,1] + -42.718;
   1:  PR[GP1:91,2] = PR[GP1:90,2] + 34.727;
   1:L PR[91] 10mm/sec CNT100;
   1:  PR[GP1:91,1] = PR[GP1:90,1] + -54.600;
   1:  PR[GP1:91,2] = PR[GP1:90,2] + 31.018;
   1:L PR[91] 10mm/sec CNT100;
   1:  PR[GP1:91,1] = PR[GP1:90,1] + -56.145;
   1:  PR[GP1:91,2] = PR[GP1:90,2] + 29.889;
   1:L PR[91] 10mm/sec CNT100;
   1:  PR[GP1:91,1] = PR[GP1:90,1] + -64.518;
   1:  PR[GP1:91,2] = PR[GP1:90,2] + 23.375;
   1:L PR[91] 10mm/sec CNT100;
   1:  PR[GP1:91,1] = PR[GP1:90,1] + -66.337;
   1:  PR[GP1:91,2] = PR[GP1:90,2] + 20.506;
   1:L PR[91] 10mm/sec CNT100;
   1:  PR[GP1:91,1] = PR[GP1:90,1] + -71.113;
   1:  PR[GP1:91,2] = PR[GP1:90,2] + 12.650;
   1:L PR[91] 10mm/sec CNT100;
   1:  PR[GP1:91,1] = PR[GP1:90,1] + -71.923;
   1:  PR[GP1:91,2] = PR[GP1:90,2] + 8.427;
   1:L PR[91] 10mm/sec CNT100;
   1:  PR[GP1:91,1] = PR[GP1:90,1] + -73.427;
   1:  PR[GP1:91,2] = PR[GP1:90,2] + 0.281;
   1:L PR[91] 10mm/sec CNT100;
   1:  PR[GP1:91,1] = PR[GP1:90,1] + -72.599;
   1:  PR[GP1:91,2] = PR[GP1:90,2] + -4.032;
   1:L PR[91] 10mm/sec CNT100;
   1:  PR[GP1:91,1] = PR[GP1:90,1] + -71.111;
   1:  PR[GP1:91,2] = PR[GP1:90,2] + -12.094;
   1:L PR[91] 10mm/sec CNT100;
   1:  PR[GP1:91,1] = PR[GP1:90,1] + -66.336;
   1:  PR[GP1:91,2] = PR[GP1:90,2] + -19.948;
   1:L PR[91] 10mm/sec CNT100;
   1:  PR[GP1:91,1] = PR[GP1:90,1] + -64.518;
   1:  PR[GP1:91,2] = PR[GP1:90,2] + -22.817;
   1:L PR[91] 10mm/sec CNT100;
   1:  PR[GP1:91,1] = PR[GP1:90,1] + -56.145;
   1:  PR[GP1:91,2] = PR[GP1:90,2] + -29.331;
   1:L PR[91] 10mm/sec CNT100;
   1:  PR[GP1:91,1] = PR[GP1:90,1] + -54.600;
   1:  PR[GP1:91,2] = PR[GP1:90,2] + -30.460;
   1:L PR[91] 10mm/sec CNT100;
   1:  PR[GP1:91,1] = PR[GP1:90,1] + -42.718;
   1:  PR[GP1:91,2] = PR[GP1:90,2] + -34.168;
   1:L PR[91] 10mm/sec CNT100;
   1:  PR[GP1:91,1] = PR[GP1:90,1] + -30.300;
   1:  PR[GP1:91,2] = PR[GP1:90,2] + -33.646;
   1:L PR[91] 10mm/sec CNT100;
   1:  PR[GP1:91,1] = PR[GP1:90,1] + -27.284;
   1:  PR[GP1:91,2] = PR[GP1:90,2] + -32.609;
   1:L PR[91] 10mm/sec CNT100;
   1:  PR[GP1:91,1] = PR[GP1:90,1] + -18.986;
   1:  PR[GP1:91,2] = PR[GP1:90,2] + -29.147;
   1:L PR[91] 10mm/sec CNT100;
   1:  PR[GP1:91,1] = PR[GP1:90,1] + -14.096;
   1:  PR[GP1:91,2] = PR[GP1:90,2] + -25.243;
   1:L PR[91] 10mm/sec CNT100;
   1:  PR[GP1:91,1] = PR[GP1:90,1] + -9.948;
   1:  PR[GP1:91,2] = PR[GP1:90,2] + -21.344;
   1:L PR[91] 10mm/sec CNT100;
   1:  PR[GP1:91,1] = PR[GP1:90,1] + -5.504;
   1:  PR[GP1:91,2] = PR[GP1:90,2] + -14.000;
   1:L PR[91] 10mm/sec CNT100;
   1:  PR[GP1:91,1] = PR[GP1:90,1] + -3.876;
   1:  PR[GP1:91,2] = PR[GP1:90,2] + -10.608;
   1:L PR[91] 10mm/sec CNT100;
   1:  PR[GP1:91,1] = PR[GP1:90,1] + 3.348;
   1:L PR[91] 10mm/sec CNT100;
   1:  PR[GP1:91,1] = PR[GP1:90,1] + 4.361;
   1:  PR[GP1:91,2] = PR[GP1:90,2] + -13.247;
   1:  PR[GP1:91,3] = PR[GP1:90,3] + 28.365;
   1:L PR[91] 10mm/sec CNT100;
   1:  PR[GP1:91,1] = PR[GP1:90,1] + 9.402;
   1:  PR[GP1:91,2] = PR[GP1:90,2] + -21.563;
   1:L PR[91] 10mm/sec CNT100;
   1:  PR[GP1:91,1] = PR[GP1:90,1] + 12.686;
   1:  PR[GP1:91,2] = PR[GP1:90,2] + -24.658;
   1:L PR[91] 10mm/sec CNT100;
   1:  PR[GP1:91,1] = PR[GP1:90,1] + 18.467;
   1:  PR[GP1:91,2] = PR[GP1:90,2] + -29.284;
   1:L PR[91] 10mm/sec CNT100;
   1:  PR[GP1:91,1] = PR[GP1:90,1] + 25.718;
   1:  PR[GP1:91,2] = PR[GP1:90,2] + -32.308;
   1:L PR[91] 10mm/sec CNT100;
   1:  PR[GP1:91,1] = PR[GP1:90,1] + 29.773;
   1:  PR[GP1:91,2] = PR[GP1:90,2] + -33.703;
   1:L PR[91] 10mm/sec CNT100;
   1:  PR[GP1:91,1] = PR[GP1:90,1] + 41.036;
   1:  PR[GP1:91,2] = PR[GP1:90,2] + -34.190;
   1:L PR[91] 10mm/sec CNT100;
   1:  PR[GP1:91,1] = PR[GP1:90,1] + 42.146;
   1:  PR[GP1:91,2] = PR[GP1:90,2] + -34.182;
   1:L PR[91] 10mm/sec CNT100;
   1:  PR[GP1:91,1] = PR[GP1:90,1] + 47.459;
   1:  PR[GP1:91,2] = PR[GP1:90,2] + -32.496;
   1:L PR[91] 10mm/sec CNT100;
   1:  PR[GP1:91,1] = PR[GP1:90,1] + 54.065;
   1:  PR[GP1:91,2] = PR[GP1:90,2] + -30.439;
   1:L PR[91] 10mm/sec CNT100;
   1:  PR[GP1:91,1] = PR[GP1:90,1] + 54.954;
   1:  PR[GP1:91,2] = PR[GP1:90,2] + -29.789;
   1:L PR[91] 10mm/sec CNT100;
   1:  PR[GP1:91,1] = PR[GP1:90,1] + 63.954;
   1:  PR[GP1:91,2] = PR[GP1:90,2] + -22.788;
   1:L PR[91] 10mm/sec CNT100;
   1:  PR[GP1:91,1] = PR[GP1:90,1] + 65.373;
   1:  PR[GP1:91,2] = PR[GP1:90,2] + -20.549;
   1:L PR[91] 10mm/sec CNT100;
   1:  PR[GP1:91,1] = PR[GP1:90,1] + 70.528;
   1:  PR[GP1:91,2] = PR[GP1:90,2] + -12.082;
   1:L PR[91] 10mm/sec CNT100;
   1:  PR[GP1:91,1] = PR[GP1:90,1] + 71.203;
   1:  PR[GP1:91,2] = PR[GP1:90,2] + -8.562;
   1:L PR[91] 10mm/sec CNT100;
   1:  PR[GP1:91,1] = PR[GP1:90,1] + 72.834;
   1:  PR[GP1:91,2] = PR[GP1:90,2] + 0.277;
   1:L PR[91] 10mm/sec CNT100;
   1:  PR[GP1:91,1] = PR[GP1:90,1] + 72.132;
   1:  PR[GP1:91,2] = PR[GP1:90,2] + 3.935;
   1:L PR[91] 10mm/sec CNT100;
   1:  PR[GP1:91,1] = PR[GP1:90,1] + 70.527;
   1:  PR[GP1:91,2] = PR[GP1:90,2] + 12.642;
   1:L PR[91] 10mm/sec CNT100;
   1:  PR[GP1:91,1] = PR[GP1:90,1] + 65.373;
   1:  PR[GP1:91,2] = PR[GP1:90,2] + 21.107;
   1:L PR[91] 10mm/sec CNT100;
   1:  PR[GP1:91,1] = PR[GP1:90,1] + 63.954;
   1:  PR[GP1:91,2] = PR[GP1:90,2] + 23.346;
   1:L PR[91] 10mm/sec CNT100;
   1:  PR[GP1:91,1] = PR[GP1:90,1] + 54.954;
   1:  PR[GP1:91,2] = PR[GP1:90,2] + 30.347;
   1:L PR[91] 10mm/sec CNT100;
   1:  PR[GP1:91,1] = PR[GP1:90,1] + 54.065;
   1:  PR[GP1:91,2] = PR[GP1:90,2] + 30.997;
   1:L PR[91] 10mm/sec CNT100;
   1:  PR[GP1:91,1] = PR[GP1:90,1] + 47.459;
   1:  PR[GP1:91,2] = PR[GP1:90,2] + 33.054;
   1:L PR[91] 10mm/sec CNT100;
   1:  PR[GP1:91,1] = PR[GP1:90,1] + 42.146;
   1:  PR[GP1:91,2] = PR[GP1:90,2] + 34.740;
   1:L PR[91] 10mm/sec CNT100;
   1:  PR[GP1:91,1] = PR[GP1:90,1] + 41.036;
   1:  PR[GP1:91,2] = PR[GP1:90,2] + 34.748;
   1:L PR[91] 10mm/sec CNT100;
   1:  PR[GP1:91,1] = PR[GP1:90,1] + 29.773;
   1:  PR[GP1:91,2] = PR[GP1:90,2] + 34.261;
   1:L PR[91] 10mm/sec CNT100;
   1:  PR[GP1:91,1] = PR[GP1:90,1] + 25.718;
   1:  PR[GP1:91,2] = PR[GP1:90,2] + 32.867;
   1:L PR[91] 10mm/sec CNT100;
   1:  PR[GP1:91,1] = PR[GP1:90,1] + 18.467;
   1:  PR[GP1:91,2] = PR[GP1:90,2] + 29.842;
   1:L PR[91] 10mm/sec CNT100;
   1:  PR[GP1:91,1] = PR[GP1:90,1] + 12.686;
   1:  PR[GP1:91,2] = PR[GP1:90,2] + 25.216;
   1:L PR[91] 10mm/sec CNT100;
   1:  PR[GP1:91,1] = PR[GP1:90,1] + 9.402;
   1:  PR[GP1:91,2] = PR[GP1:90,2] + 22.121;
   1:L PR[91] 10mm/sec CNT100;
   1:  PR[GP1:91,1] = PR[GP1:90,1] + 4.362;
   1:  PR[GP1:91,2] = PR[GP1:90,2] + 13.806;
   1:L PR[91] 10mm/sec CNT100;
   1:  PR[GP1:91,1] = PR[GP1:90,1] + 3.249;
   1:  PR[GP1:91,2] = PR[GP1:90,2] + 11.491;
   1:L PR[91] 10mm/sec CNT100;
   1:  PR[GP1:91,1] = PR[GP1:90,1] + -3.787;
   1:L PR[91] 10mm/sec CNT100;
   1:  PR[GP1:91,1] = PR[GP1:90,1] + -4.897;
   1:  PR[GP1:91,2] = PR[GP1:90,2] + 13.812;
   1:L PR[91] 10mm/sec CNT100;
   1:  PR[GP1:91,1] = PR[GP1:90,1] + -9.935;
   1:  PR[GP1:91,2] = PR[GP1:90,2] + 22.139;
   1:L PR[91] 10mm/sec CNT100;
   1:  PR[GP1:91,1] = PR[GP1:90,1] + -13.222;
   1:  PR[GP1:91,2] = PR[GP1:90,2] + 25.228;
   1:L PR[91] 10mm/sec CNT100;
   1:  PR[GP1:91,1] = PR[GP1:90,1] + -19.003;
   1:  PR[GP1:91,2] = PR[GP1:90,2] + 29.844;
   1:L PR[91] 10mm/sec CNT100;
   1:  PR[GP1:91,1] = PR[GP1:90,1] + -26.257;
   1:  PR[GP1:91,2] = PR[GP1:90,2] + 32.870;
   1:L PR[91] 10mm/sec CNT100;
   1:  PR[GP1:91,1] = PR[GP1:90,1] + -30.310;
   1:  PR[GP1:91,2] = PR[GP1:90,2] + 34.264;
   1:L PR[91] 10mm/sec CNT100;
   1:  PR[GP1:91,1] = PR[GP1:90,1] + -41.575;
   1:  PR[GP1:91,2] = PR[GP1:90,2] + 34.747;
   1:L PR[91] 10mm/sec CNT100;
   1:  PR[GP1:91,1] = PR[GP1:90,1] + -42.682;
   1:  PR[GP1:91,2] = PR[GP1:90,2] + 34.738;
   1:L PR[91] 10mm/sec CNT100;
   1:  PR[GP1:91,1] = PR[GP1:90,1] + -47.986;
   1:  PR[GP1:91,2] = PR[GP1:90,2] + 33.054;
   1:L PR[91] 10mm/sec CNT100;
   1:  PR[GP1:91,1] = PR[GP1:90,1] + -54.598;
   1:  PR[GP1:91,2] = PR[GP1:90,2] + 30.993;
   1:L PR[91] 10mm/sec CNT100;
   1:  PR[GP1:91,1] = PR[GP1:90,1] + -55.488;
   1:  PR[GP1:91,2] = PR[GP1:90,2] + 30.342;
   1:L PR[91] 10mm/sec CNT100;
   1:  PR[GP1:91,1] = PR[GP1:90,1] + -64.483;
   1:  PR[GP1:91,2] = PR[GP1:90,2] + 23.345;
   1:L PR[91] 10mm/sec CNT100;
   1:  PR[GP1:91,1] = PR[GP1:90,1] + -65.902;
   1:  PR[GP1:91,2] = PR[GP1:90,2] + 21.106;
   1:L PR[91] 10mm/sec CNT100;
   1:  PR[GP1:91,1] = PR[GP1:90,1] + -71.055;
   1:  PR[GP1:91,2] = PR[GP1:90,2] + 12.630;
   1:L PR[91] 10mm/sec CNT100;
   1:  PR[GP1:91,1] = PR[GP1:90,1] + -71.730;
   1:  PR[GP1:91,2] = PR[GP1:90,2] + 9.111;
   1:L PR[91] 10mm/sec CNT100;
   1:  PR[GP1:91,1] = PR[GP1:90,1] + -73.361;
   1:  PR[GP1:91,2] = PR[GP1:90,2] + 0.281;
   1:L PR[91] 10mm/sec CNT100;
   1:  PR[GP1:91,1] = PR[GP1:90,1] + -72.658;
   1:  PR[GP1:91,2] = PR[GP1:90,2] + -3.376;
   1:L PR[91] 10mm/sec CNT100;
   1:  PR[GP1:91,1] = PR[GP1:90,1] + -71.054;
   1:  PR[GP1:91,2] = PR[GP1:90,2] + -12.074;
   1:L PR[91] 10mm/sec CNT100;
   1:  PR[GP1:91,1] = PR[GP1:90,1] + -65.902;
   1:  PR[GP1:91,2] = PR[GP1:90,2] + -20.548;
   1:L PR[91] 10mm/sec CNT100;
   1:  PR[GP1:91,1] = PR[GP1:90,1] + -64.483;
   1:  PR[GP1:91,2] = PR[GP1:90,2] + -22.787;
   1:L PR[91] 10mm/sec CNT100;
   1:  PR[GP1:91,1] = PR[GP1:90,1] + -55.488;
   1:  PR[GP1:91,2] = PR[GP1:90,2] + -29.784;
   1:L PR[91] 10mm/sec CNT100;
   1:  PR[GP1:91,1] = PR[GP1:90,1] + -54.598;
   1:  PR[GP1:91,2] = PR[GP1:90,2] + -30.435;
   1:L PR[91] 10mm/sec CNT100;
   1:  PR[GP1:91,1] = PR[GP1:90,1] + -47.986;
   1:  PR[GP1:91,2] = PR[GP1:90,2] + -32.496;
   1:L PR[91] 10mm/sec CNT100;
   1:  PR[GP1:91,1] = PR[GP1:90,1] + -42.682;
   1:  PR[GP1:91,2] = PR[GP1:90,2] + -34.180;
   1:L PR[91] 10mm/sec CNT100;
   1:  PR[GP1:91,1] = PR[GP1:90,1] + -41.574;
   1:  PR[GP1:91,2] = PR[GP1:90,2] + -34.189;
   1:L PR[91] 10mm/sec CNT100;
   1:  PR[GP1:91,1] = PR[GP1:90,1] + -30.310;
   1:  PR[GP1:91,2] = PR[GP1:90,2] + -33.706;
   1:L PR[91] 10mm/sec CNT100;
   1:  PR[GP1:91,1] = PR[GP1:90,1] + -26.257;
   1:  PR[GP1:91,2] = PR[GP1:90,2] + -32.312;
   1:L PR[91] 10mm/sec CNT100;
   1:  PR[GP1:91,1] = PR[GP1:90,1] + -19.003;
   1:  PR[GP1:91,2] = PR[GP1:90,2] + -29.286;
   1:L PR[91] 10mm/sec CNT100;
   1:  PR[GP1:91,1] = PR[GP1:90,1] + -13.222;
   1:  PR[GP1:91,2] = PR[GP1:90,2] + -24.670;
   1:L PR[91] 10mm/sec CNT100;
   1:  PR[GP1:91,1] = PR[GP1:90,1] + -9.936;
   1:  PR[GP1:91,2] = PR[GP1:90,2] + -21.581;
   1:L PR[91] 10mm/sec CNT100;
   1:  PR[GP1:91,1] = PR[GP1:90,1] + -4.897;
   1:  PR[GP1:91,2] = PR[GP1:90,2] + -13.255;
   1:L PR[91] 10mm/sec CNT100;
   1:  PR[GP1:91,1] = PR[GP1:90,1] + -3.783;
   1:  PR[GP1:91,2] = PR[GP1:90,2] + -10.933;
   1:L PR[91] 10mm/sec CNT100;
   1:  PR[GP1:91,1] = PR[GP1:90,1] + 3.253;
   1:L PR[91] 10mm/sec CNT100;
   1:  PR[GP1:91,1] = PR[GP1:90,1] + 3.754;
   1:  PR[GP1:91,2] = PR[GP1:90,2] + -12.505;
   1:  PR[GP1:91,3] = PR[GP1:90,3] + 28.975;
   1:L PR[91] 10mm/sec CNT100;
   1:  PR[GP1:91,1] = PR[GP1:90,1] + 9.390;
   1:  PR[GP1:91,2] = PR[GP1:90,2] + -21.801;
   1:L PR[91] 10mm/sec CNT100;
   1:  PR[GP1:91,1] = PR[GP1:90,1] + 11.813;
   1:  PR[GP1:91,2] = PR[GP1:90,2] + -24.084;
   1:L PR[91] 10mm/sec CNT100;
   1:  PR[GP1:91,1] = PR[GP1:90,1] + 18.485;
   1:  PR[GP1:91,2] = PR[GP1:90,2] + -29.423;
   1:L PR[91] 10mm/sec CNT100;
   1:  PR[GP1:91,1] = PR[GP1:90,1] + 24.692;
   1:  PR[GP1:91,2] = PR[GP1:90,2] + -32.012;
   1:L PR[91] 10mm/sec CNT100;
   1:  PR[GP1:91,1] = PR[GP1:90,1] + 29.784;
   1:  PR[GP1:91,2] = PR[GP1:90,2] + -33.763;
   1:L PR[91] 10mm/sec CNT100;
   1:  PR[GP1:91,1] = PR[GP1:90,1] + 40.001;
   1:  PR[GP1:91,2] = PR[GP1:90,2] + -34.205;
   1:L PR[91] 10mm/sec CNT100;
   1:  PR[GP1:91,1] = PR[GP1:90,1] + 42.128;
   1:  PR[GP1:91,2] = PR[GP1:90,2] + -34.188;
   1:L PR[91] 10mm/sec CNT100;
   1:  PR[GP1:91,1] = PR[GP1:90,1] + 51.952;
   1:  PR[GP1:91,2] = PR[GP1:90,2] + -31.071;
   1:L PR[91] 10mm/sec CNT100;
   1:  PR[GP1:91,1] = PR[GP1:90,1] + 54.063;
   1:  PR[GP1:91,2] = PR[GP1:90,2] + -30.414;
   1:L PR[91] 10mm/sec CNT100;
   1:  PR[GP1:91,1] = PR[GP1:90,1] + 54.297;
   1:  PR[GP1:91,2] = PR[GP1:90,2] + -30.243;
   1:L PR[91] 10mm/sec CNT100;
   1:  PR[GP1:91,1] = PR[GP1:90,1] + 63.918;
   1:  PR[GP1:91,2] = PR[GP1:90,2] + -22.757;
   1:L PR[91] 10mm/sec CNT100;
   1:  PR[GP1:91,1] = PR[GP1:90,1] + 64.938;
   1:  PR[GP1:91,2] = PR[GP1:90,2] + -21.149;
   1:L PR[91] 10mm/sec CNT100;
   1:  PR[GP1:91,1] = PR[GP1:90,1] + 70.470;
   1:  PR[GP1:91,2] = PR[GP1:90,2] + -12.063;
   1:L PR[91] 10mm/sec CNT100;
   1:  PR[GP1:91,1] = PR[GP1:90,1] + 71.010;
   1:  PR[GP1:91,2] = PR[GP1:90,2] + -9.248;
   1:L PR[91] 10mm/sec CNT100;
   1:  PR[GP1:91,1] = PR[GP1:90,1] + 72.768;
   1:  PR[GP1:91,2] = PR[GP1:90,2] + 0.277;
   1:L PR[91] 10mm/sec CNT100;
   1:  PR[GP1:91,1] = PR[GP1:90,1] + 72.191;
   1:  PR[GP1:91,2] = PR[GP1:90,2] + 3.279;
   1:L PR[91] 10mm/sec CNT100;
   1:  PR[GP1:91,1] = PR[GP1:90,1] + 70.469;
   1:  PR[GP1:91,2] = PR[GP1:90,2] + 12.623;
   1:L PR[91] 10mm/sec CNT100;
   1:  PR[GP1:91,1] = PR[GP1:90,1] + 64.938;
   1:  PR[GP1:91,2] = PR[GP1:90,2] + 21.707;
   1:L PR[91] 10mm/sec CNT100;
   1:  PR[GP1:91,1] = PR[GP1:90,1] + 63.918;
   1:  PR[GP1:91,2] = PR[GP1:90,2] + 23.316;
   1:L PR[91] 10mm/sec CNT100;
   1:  PR[GP1:91,1] = PR[GP1:90,1] + 54.297;
   1:  PR[GP1:91,2] = PR[GP1:90,2] + 30.801;
   1:L PR[91] 10mm/sec CNT100;
   1:  PR[GP1:91,1] = PR[GP1:90,1] + 54.063;
   1:  PR[GP1:91,2] = PR[GP1:90,2] + 30.972;
   1:L PR[91] 10mm/sec CNT100;
   1:  PR[GP1:91,1] = PR[GP1:90,1] + 51.952;
   1:  PR[GP1:91,2] = PR[GP1:90,2] + 31.629;
   1:L PR[91] 10mm/sec CNT100;
   1:  PR[GP1:91,1] = PR[GP1:90,1] + 42.128;
   1:  PR[GP1:91,2] = PR[GP1:90,2] + 34.746;
   1:L PR[91] 10mm/sec CNT100;
   1:  PR[GP1:91,1] = PR[GP1:90,1] + 40.001;
   1:  PR[GP1:91,2] = PR[GP1:90,2] + 34.763;
   1:L PR[91] 10mm/sec CNT100;
   1:  PR[GP1:91,1] = PR[GP1:90,1] + 29.784;
   1:  PR[GP1:91,2] = PR[GP1:90,2] + 34.321;
   1:L PR[91] 10mm/sec CNT100;
   1:  PR[GP1:91,1] = PR[GP1:90,1] + 24.692;
   1:  PR[GP1:91,2] = PR[GP1:90,2] + 32.570;
   1:L PR[91] 10mm/sec CNT100;
   1:  PR[GP1:91,1] = PR[GP1:90,1] + 18.485;
   1:  PR[GP1:91,2] = PR[GP1:90,2] + 29.981;
   1:L PR[91] 10mm/sec CNT100;
   1:  PR[GP1:91,1] = PR[GP1:90,1] + 11.813;
   1:  PR[GP1:91,2] = PR[GP1:90,2] + 24.643;
   1:L PR[91] 10mm/sec CNT100;
   1:  PR[GP1:91,1] = PR[GP1:90,1] + 9.390;
   1:  PR[GP1:91,2] = PR[GP1:90,2] + 22.359;
   1:L PR[91] 10mm/sec CNT100;
   1:  PR[GP1:91,1] = PR[GP1:90,1] + 3.755;
   1:  PR[GP1:91,2] = PR[GP1:90,2] + 13.064;
   1:L PR[91] 10mm/sec CNT100;
   1:  PR[GP1:91,1] = PR[GP1:90,1] + 3.155;
   1:  PR[GP1:91,2] = PR[GP1:90,2] + 11.816;
   1:L PR[91] 10mm/sec CNT100;
   1:  PR[GP1:91,1] = PR[GP1:90,1] + -3.692;
   1:L PR[91] 10mm/sec CNT100;
   1:  PR[GP1:91,1] = PR[GP1:90,1] + -4.290;
   1:  PR[GP1:91,2] = PR[GP1:90,2] + 13.067;
   1:L PR[91] 10mm/sec CNT100;
   1:  PR[GP1:91,1] = PR[GP1:90,1] + -9.923;
   1:  PR[GP1:91,2] = PR[GP1:90,2] + 22.375;
   1:L PR[91] 10mm/sec CNT100;
   1:  PR[GP1:91,1] = PR[GP1:90,1] + -12.348;
   1:  PR[GP1:91,2] = PR[GP1:90,2] + 24.655;
   1:L PR[91] 10mm/sec CNT100;
   1:  PR[GP1:91,1] = PR[GP1:90,1] + -19.020;
   1:  PR[GP1:91,2] = PR[GP1:90,2] + 29.983;
   1:L PR[91] 10mm/sec CNT100;
   1:  PR[GP1:91,1] = PR[GP1:90,1] + -25.230;
   1:  PR[GP1:91,2] = PR[GP1:90,2] + 32.573;
   1:L PR[91] 10mm/sec CNT100;
   1:  PR[GP1:91,1] = PR[GP1:90,1] + -30.320;
   1:  PR[GP1:91,2] = PR[GP1:90,2] + 34.324;
   1:L PR[91] 10mm/sec CNT100;
   1:  PR[GP1:91,1] = PR[GP1:90,1] + -40.539;
   1:  PR[GP1:91,2] = PR[GP1:90,2] + 34.762;
   1:L PR[91] 10mm/sec CNT100;
   1:  PR[GP1:91,1] = PR[GP1:90,1] + -42.664;
   1:  PR[GP1:91,2] = PR[GP1:90,2] + 34.745;
   1:L PR[91] 10mm/sec CNT100;
   1:  PR[GP1:91,1] = PR[GP1:90,1] + -52.478;
   1:  PR[GP1:91,2] = PR[GP1:90,2] + 31.628;
   1:L PR[91] 10mm/sec CNT100;
   1:  PR[GP1:91,1] = PR[GP1:90,1] + -54.596;
   1:  PR[GP1:91,2] = PR[GP1:90,2] + 30.967;
   1:L PR[91] 10mm/sec CNT100;
   1:  PR[GP1:91,1] = PR[GP1:90,1] + -54.830;
   1:  PR[GP1:91,2] = PR[GP1:90,2] + 30.796;
   1:L PR[91] 10mm/sec CNT100;
   1:  PR[GP1:91,1] = PR[GP1:90,1] + -64.448;
   1:  PR[GP1:91,2] = PR[GP1:90,2] + 23.315;
   1:L PR[91] 10mm/sec CNT100;
   1:  PR[GP1:91,1] = PR[GP1:90,1] + -65.468;
   1:  PR[GP1:91,2] = PR[GP1:90,2] + 21.706;
   1:L PR[91] 10mm/sec CNT100;
   1:  PR[GP1:91,1] = PR[GP1:90,1] + -70.997;
   1:  PR[GP1:91,2] = PR[GP1:90,2] + 12.610;
   1:L PR[91] 10mm/sec CNT100;
   1:  PR[GP1:91,1] = PR[GP1:90,1] + -71.537;
   1:  PR[GP1:91,2] = PR[GP1:90,2] + 9.795;
   1:L PR[91] 10mm/sec CNT100;
   1:  PR[GP1:91,1] = PR[GP1:90,1] + -73.294;
   1:  PR[GP1:91,2] = PR[GP1:90,2] + 0.281;
   1:L PR[91] 10mm/sec CNT100;
   1:  PR[GP1:91,1] = PR[GP1:90,1] + -72.718;
   1:  PR[GP1:91,2] = PR[GP1:90,2] + -2.720;
   1:L PR[91] 10mm/sec CNT100;
   1:  PR[GP1:91,1] = PR[GP1:90,1] + -70.996;
   1:  PR[GP1:91,2] = PR[GP1:90,2] + -12.054;
   1:L PR[91] 10mm/sec CNT100;
   1:  PR[GP1:91,1] = PR[GP1:90,1] + -65.467;
   1:  PR[GP1:91,2] = PR[GP1:90,2] + -21.148;
   1:L PR[91] 10mm/sec CNT100;
   1:  PR[GP1:91,1] = PR[GP1:90,1] + -64.448;
   1:  PR[GP1:91,2] = PR[GP1:90,2] + -22.757;
   1:L PR[91] 10mm/sec CNT100;
   1:  PR[GP1:91,1] = PR[GP1:90,1] + -54.830;
   1:  PR[GP1:91,2] = PR[GP1:90,2] + -30.238;
   1:L PR[91] 10mm/sec CNT100;
   1:  PR[GP1:91,1] = PR[GP1:90,1] + -54.596;
   1:  PR[GP1:91,2] = PR[GP1:90,2] + -30.409;
   1:L PR[91] 10mm/sec CNT100;
   1:  PR[GP1:91,1] = PR[GP1:90,1] + -52.478;
   1:  PR[GP1:91,2] = PR[GP1:90,2] + -31.069;
   1:L PR[91] 10mm/sec CNT100;
   1:  PR[GP1:91,1] = PR[GP1:90,1] + -42.663;
   1:  PR[GP1:91,2] = PR[GP1:90,2] + -34.187;
   1:L PR[91] 10mm/sec CNT100;
   1:  PR[GP1:91,1] = PR[GP1:90,1] + -40.539;
   1:  PR[GP1:91,2] = PR[GP1:90,2] + -34.204;
   1:L PR[91] 10mm/sec CNT100;
   1:  PR[GP1:91,1] = PR[GP1:90,1] + -30.320;
   1:  PR[GP1:91,2] = PR[GP1:90,2] + -33.766;
   1:L PR[91] 10mm/sec CNT100;
   1:  PR[GP1:91,1] = PR[GP1:90,1] + -25.230;
   1:  PR[GP1:91,2] = PR[GP1:90,2] + -32.015;
   1:L PR[91] 10mm/sec CNT100;
   1:  PR[GP1:91,1] = PR[GP1:90,1] + -19.020;
   1:  PR[GP1:91,2] = PR[GP1:90,2] + -29.425;
   1:L PR[91] 10mm/sec CNT100;
   1:  PR[GP1:91,1] = PR[GP1:90,1] + -12.348;
   1:  PR[GP1:91,2] = PR[GP1:90,2] + -24.097;
   1:L PR[91] 10mm/sec CNT100;
   1:  PR[GP1:91,1] = PR[GP1:90,1] + -9.923;
   1:  PR[GP1:91,2] = PR[GP1:90,2] + -21.817;
   1:L PR[91] 10mm/sec CNT100;
   1:  PR[GP1:91,1] = PR[GP1:90,1] + -4.291;
   1:  PR[GP1:91,2] = PR[GP1:90,2] + -12.510;
   1:L PR[91] 10mm/sec CNT100;
   1:  PR[GP1:91,1] = PR[GP1:90,1] + -3.689;
   1:  PR[GP1:91,2] = PR[GP1:90,2] + -11.258;
   1:L PR[91] 10mm/sec CNT100;
   1:  PR[GP1:91,1] = PR[GP1:90,1] + 3.157;
   1:L PR[91] 10mm/sec CNT100;
   1:  PR[GP1:91,1] = PR[GP1:90,1] + 3.591;
   1:  PR[GP1:91,2] = PR[GP1:90,2] + -12.493;
   1:  PR[GP1:91,3] = PR[GP1:90,3] + 29.585;
   1:L PR[91] 10mm/sec CNT100;
   1:  PR[GP1:91,1] = PR[GP1:90,1] + 9.377;
   1:  PR[GP1:91,2] = PR[GP1:90,2] + -22.039;
   1:L PR[91] 10mm/sec CNT100;
   1:  PR[GP1:91,1] = PR[GP1:90,1] + 10.939;
   1:  PR[GP1:91,2] = PR[GP1:90,2] + -23.511;
   1:L PR[91] 10mm/sec CNT100;
   1:  PR[GP1:91,1] = PR[GP1:90,1] + 18.503;
   1:  PR[GP1:91,2] = PR[GP1:90,2] + -29.562;
   1:L PR[91] 10mm/sec CNT100;
   1:  PR[GP1:91,1] = PR[GP1:90,1] + 23.666;
   1:  PR[GP1:91,2] = PR[GP1:90,2] + -31.716;
   1:L PR[91] 10mm/sec CNT100;
   1:  PR[GP1:91,1] = PR[GP1:90,1] + 29.794;
   1:  PR[GP1:91,2] = PR[GP1:90,2] + -33.823;
   1:L PR[91] 10mm/sec CNT100;
   1:  PR[GP1:91,1] = PR[GP1:90,1] + 38.966;
   1:  PR[GP1:91,2] = PR[GP1:90,2] + -34.220;
   1:L PR[91] 10mm/sec CNT100;
   1:  PR[GP1:91,1] = PR[GP1:90,1] + 42.109;
   1:  PR[GP1:91,2] = PR[GP1:90,2] + -34.195;
   1:L PR[91] 10mm/sec CNT100;
   1:  PR[GP1:91,1] = PR[GP1:90,1] + 53.674;
   1:  PR[GP1:91,2] = PR[GP1:90,2] + -30.525;
   1:L PR[91] 10mm/sec CNT100;
   1:  PR[GP1:91,1] = PR[GP1:90,1] + 54.014;
   1:  PR[GP1:91,2] = PR[GP1:90,2] + -30.402;
   1:L PR[91] 10mm/sec CNT100;
   1:  PR[GP1:91,1] = PR[GP1:90,1] + 63.883;
   1:  PR[GP1:91,2] = PR[GP1:90,2] + -22.727;
   1:L PR[91] 10mm/sec CNT100;
   1:  PR[GP1:91,1] = PR[GP1:90,1] + 64.504;
   1:  PR[GP1:91,2] = PR[GP1:90,2] + -21.749;
   1:L PR[91] 10mm/sec CNT100;
   1:  PR[GP1:91,1] = PR[GP1:90,1] + 70.412;
   1:  PR[GP1:91,2] = PR[GP1:90,2] + -12.044;
   1:L PR[91] 10mm/sec CNT100;
   1:  PR[GP1:91,1] = PR[GP1:90,1] + 70.817;
   1:  PR[GP1:91,2] = PR[GP1:90,2] + -9.933;
   1:L PR[91] 10mm/sec CNT100;
   1:  PR[GP1:91,1] = PR[GP1:90,1] + 72.702;
   1:  PR[GP1:91,2] = PR[GP1:90,2] + 0.277;
   1:L PR[91] 10mm/sec CNT100;
   1:  PR[GP1:91,1] = PR[GP1:90,1] + 72.251;
   1:  PR[GP1:91,2] = PR[GP1:90,2] + 2.622;
   1:L PR[91] 10mm/sec CNT100;
   1:  PR[GP1:91,1] = PR[GP1:90,1] + 70.411;
   1:  PR[GP1:91,2] = PR[GP1:90,2] + 12.604;
   1:L PR[91] 10mm/sec CNT100;
   1:  PR[GP1:91,1] = PR[GP1:90,1] + 64.503;
   1:  PR[GP1:91,2] = PR[GP1:90,2] + 22.307;
   1:L PR[91] 10mm/sec CNT100;
   1:  PR[GP1:91,1] = PR[GP1:90,1] + 63.883;
   1:  PR[GP1:91,2] = PR[GP1:90,2] + 23.285;
   1:L PR[91] 10mm/sec CNT100;
   1:  PR[GP1:91,1] = PR[GP1:90,1] + 54.014;
   1:  PR[GP1:91,2] = PR[GP1:90,2] + 30.961;
   1:L PR[91] 10mm/sec CNT100;
   1:  PR[GP1:91,1] = PR[GP1:90,1] + 53.674;
   1:  PR[GP1:91,2] = PR[GP1:90,2] + 31.084;
   1:L PR[91] 10mm/sec CNT100;
   1:  PR[GP1:91,1] = PR[GP1:90,1] + 42.109;
   1:  PR[GP1:91,2] = PR[GP1:90,2] + 34.753;
   1:L PR[91] 10mm/sec CNT100;
   1:  PR[GP1:91,1] = PR[GP1:90,1] + 38.966;
   1:  PR[GP1:91,2] = PR[GP1:90,2] + 34.778;
   1:L PR[91] 10mm/sec CNT100;
   1:  PR[GP1:91,1] = PR[GP1:90,1] + 29.794;
   1:  PR[GP1:91,2] = PR[GP1:90,2] + 34.381;
   1:L PR[91] 10mm/sec CNT100;
   1:  PR[GP1:91,1] = PR[GP1:90,1] + 23.666;
   1:  PR[GP1:91,2] = PR[GP1:90,2] + 32.274;
   1:L PR[91] 10mm/sec CNT100;
   1:  PR[GP1:91,1] = PR[GP1:90,1] + 18.503;
   1:  PR[GP1:91,2] = PR[GP1:90,2] + 30.120;
   1:L PR[91] 10mm/sec CNT100;
   1:  PR[GP1:91,1] = PR[GP1:90,1] + 10.939;
   1:  PR[GP1:91,2] = PR[GP1:90,2] + 24.069;
   1:L PR[91] 10mm/sec CNT100;
   1:  PR[GP1:91,1] = PR[GP1:90,1] + 9.378;
   1:  PR[GP1:91,2] = PR[GP1:90,2] + 22.597;
   1:L PR[91] 10mm/sec CNT100;
   1:  PR[GP1:91,1] = PR[GP1:90,1] + 3.586;
   1:  PR[GP1:91,2] = PR[GP1:90,2] + 13.043;
   1:L PR[91] 10mm/sec CNT100;
   1:  PR[GP1:91,1] = PR[GP1:90,1] + 3.012;
   1:  PR[GP1:91,2] = PR[GP1:90,2] + 12.141;
   1:L PR[91] 10mm/sec CNT100;
   1:  PR[GP1:91,1] = PR[GP1:90,1] + -3.546;
   1:L PR[91] 10mm/sec CNT100;
   1:  PR[GP1:91,1] = PR[GP1:90,1] + -4.119;
   1:  PR[GP1:91,2] = PR[GP1:90,2] + 13.043;
   1:L PR[91] 10mm/sec CNT100;
   1:  PR[GP1:91,1] = PR[GP1:90,1] + -9.910;
   1:  PR[GP1:91,2] = PR[GP1:90,2] + 22.612;
   1:L PR[91] 10mm/sec CNT100;
   1:  PR[GP1:91,1] = PR[GP1:90,1] + -11.473;
   1:  PR[GP1:91,2] = PR[GP1:90,2] + 24.082;
   1:L PR[91] 10mm/sec CNT100;
   1:  PR[GP1:91,1] = PR[GP1:90,1] + -19.037;
   1:  PR[GP1:91,2] = PR[GP1:90,2] + 30.122;
   1:L PR[91] 10mm/sec CNT100;
   1:  PR[GP1:91,1] = PR[GP1:90,1] + -24.204;
   1:  PR[GP1:91,2] = PR[GP1:90,2] + 32.277;
   1:L PR[91] 10mm/sec CNT100;
   1:  PR[GP1:91,1] = PR[GP1:90,1] + -30.330;
   1:  PR[GP1:91,2] = PR[GP1:90,2] + 34.384;
   1:L PR[91] 10mm/sec CNT100;
   1:  PR[GP1:91,1] = PR[GP1:90,1] + -39.504;
   1:  PR[GP1:91,2] = PR[GP1:90,2] + 34.777;
   1:L PR[91] 10mm/sec CNT100;
   1:  PR[GP1:91,1] = PR[GP1:90,1] + -42.645;
   1:  PR[GP1:91,2] = PR[GP1:90,2] + 34.752;
   1:L PR[91] 10mm/sec CNT100;
   1:  PR[GP1:91,1] = PR[GP1:90,1] + -54.208;
   1:  PR[GP1:91,2] = PR[GP1:90,2] + 31.079;
   1:L PR[91] 10mm/sec CNT100;
   1:  PR[GP1:91,1] = PR[GP1:90,1] + -54.547;
   1:  PR[GP1:91,2] = PR[GP1:90,2] + 30.956;
   1:L PR[91] 10mm/sec CNT100;
   1:  PR[GP1:91,1] = PR[GP1:90,1] + -64.413;
   1:  PR[GP1:91,2] = PR[GP1:90,2] + 23.285;
   1:L PR[91] 10mm/sec CNT100;
   1:  PR[GP1:91,1] = PR[GP1:90,1] + -65.033;
   1:  PR[GP1:91,2] = PR[GP1:90,2] + 22.306;
   1:L PR[91] 10mm/sec CNT100;
   1:  PR[GP1:91,1] = PR[GP1:90,1] + -70.939;
   1:  PR[GP1:91,2] = PR[GP1:90,2] + 12.591;
   1:L PR[91] 10mm/sec CNT100;
   1:  PR[GP1:91,1] = PR[GP1:90,1] + -71.344;
   1:  PR[GP1:91,2] = PR[GP1:90,2] + 10.480;
   1:L PR[91] 10mm/sec CNT100;
   1:  PR[GP1:91,1] = PR[GP1:90,1] + -73.228;
   1:  PR[GP1:91,2] = PR[GP1:90,2] + 0.281;
   1:L PR[91] 10mm/sec CNT100;
   1:  PR[GP1:91,1] = PR[GP1:90,1] + -72.777;
   1:  PR[GP1:91,2] = PR[GP1:90,2] + -2.063;
   1:L PR[91] 10mm/sec CNT100;
   1:  PR[GP1:91,1] = PR[GP1:90,1] + -70.938;
   1:  PR[GP1:91,2] = PR[GP1:90,2] + -12.035;
   1:L PR[91] 10mm/sec CNT100;
   1:  PR[GP1:91,1] = PR[GP1:90,1] + -65.033;
   1:  PR[GP1:91,2] = PR[GP1:90,2] + -21.748;
   1:L PR[91] 10mm/sec CNT100;
   1:  PR[GP1:91,1] = PR[GP1:90,1] + -64.413;
   1:  PR[GP1:91,2] = PR[GP1:90,2] + -22.727;
   1:L PR[91] 10mm/sec CNT100;
   1:  PR[GP1:91,1] = PR[GP1:90,1] + -56.784;
   1:  PR[GP1:91,2] = PR[GP1:90,2] + -28.660;
   1:L PR[91] 10mm/sec CNT100;
   1:  PR[GP1:91,1] = PR[GP1:90,1] + -54.547;
   1:  PR[GP1:91,2] = PR[GP1:90,2] + -30.398;
   1:L PR[91] 10mm/sec CNT100;
   1:  PR[GP1:91,1] = PR[GP1:90,1] + -54.208;
   1:  PR[GP1:91,2] = PR[GP1:90,2] + -30.521;
   1:L PR[91] 10mm/sec CNT100;
   1:  PR[GP1:91,1] = PR[GP1:90,1] + -42.644;
   1:  PR[GP1:91,2] = PR[GP1:90,2] + -34.194;
   1:L PR[91] 10mm/sec CNT100;
   1:  PR[GP1:91,1] = PR[GP1:90,1] + -39.504;
   1:  PR[GP1:91,2] = PR[GP1:90,2] + -34.219;
   1:L PR[91] 10mm/sec CNT100;
   1:  PR[GP1:91,1] = PR[GP1:90,1] + -30.330;
   1:  PR[GP1:91,2] = PR[GP1:90,2] + -33.826;
   1:L PR[91] 10mm/sec CNT100;
   1:  PR[GP1:91,1] = PR[GP1:90,1] + -24.204;
   1:  PR[GP1:91,2] = PR[GP1:90,2] + -31.719;
   1:L PR[91] 10mm/sec CNT100;
   1:  PR[GP1:91,1] = PR[GP1:90,1] + -19.037;
   1:  PR[GP1:91,2] = PR[GP1:90,2] + -29.564;
   1:L PR[91] 10mm/sec CNT100;
   1:  PR[GP1:91,1] = PR[GP1:90,1] + -11.473;
   1:  PR[GP1:91,2] = PR[GP1:90,2] + -23.524;
   1:L PR[91] 10mm/sec CNT100;
   1:  PR[GP1:91,1] = PR[GP1:90,1] + -9.910;
   1:  PR[GP1:91,2] = PR[GP1:90,2] + -22.054;
   1:L PR[91] 10mm/sec CNT100;
   1:  PR[GP1:91,1] = PR[GP1:90,1] + -4.114;
   1:  PR[GP1:91,2] = PR[GP1:90,2] + -12.477;
   1:L PR[91] 10mm/sec CNT100;
   1:  PR[GP1:91,1] = PR[GP1:90,1] + -3.546;
   1:  PR[GP1:91,2] = PR[GP1:90,2] + -11.583;
   1:L PR[91] 10mm/sec CNT100;
   1:  PR[GP1:91,1] = PR[GP1:90,1] + 3.012;
   1:L PR[91] 10mm/sec CNT100;
   1:  PR[GP1:91,1] = PR[GP1:90,1] + 6.638;
   1:  PR[GP1:91,2] = PR[GP1:90,2] + -17.778;
   1:  PR[GP1:91,3] = PR[GP1:90,3] + 30.195;
   1:L PR[91] 10mm/sec CNT100;
   1:  PR[GP1:91,1] = PR[GP1:90,1] + 9.365;
   1:  PR[GP1:91,2] = PR[GP1:90,2] + -22.276;
   1:L PR[91] 10mm/sec CNT100;
   1:  PR[GP1:91,1] = PR[GP1:90,1] + 10.066;
   1:  PR[GP1:91,2] = PR[GP1:90,2] + -22.937;
   1:L PR[91] 10mm/sec CNT100;
   1:  PR[GP1:91,1] = PR[GP1:90,1] + 18.520;
   1:  PR[GP1:91,2] = PR[GP1:90,2] + -29.701;
   1:L PR[91] 10mm/sec CNT100;
   1:  PR[GP1:91,1] = PR[GP1:90,1] + 22.640;
   1:  PR[GP1:91,2] = PR[GP1:90,2] + -31.420;
   1:L PR[91] 10mm/sec CNT100;
   1:  PR[GP1:91,1] = PR[GP1:90,1] + 29.804;
   1:  PR[GP1:91,2] = PR[GP1:90,2] + -33.883;
   1:L PR[91] 10mm/sec CNT100;
   1:  PR[GP1:91,1] = PR[GP1:90,1] + 37.931;
   1:  PR[GP1:91,2] = PR[GP1:90,2] + -34.235;
   1:L PR[91] 10mm/sec CNT100;
   1:  PR[GP1:91,1] = PR[GP1:90,1] + 42.091;
   1:  PR[GP1:91,2] = PR[GP1:90,2] + -34.202;
   1:L PR[91] 10mm/sec CNT100;
   1:  PR[GP1:91,1] = PR[GP1:90,1] + 52.755;
   1:  PR[GP1:91,2] = PR[GP1:90,2] + -30.818;
   1:L PR[91] 10mm/sec CNT100;
   1:  PR[GP1:91,1] = PR[GP1:90,1] + 53.960;
   1:  PR[GP1:91,2] = PR[GP1:90,2] + -30.382;
   1:L PR[91] 10mm/sec CNT100;
   1:  PR[GP1:91,1] = PR[GP1:90,1] + 63.844;
   1:  PR[GP1:91,2] = PR[GP1:90,2] + -22.700;
   1:L PR[91] 10mm/sec CNT100;
   1:  PR[GP1:91,1] = PR[GP1:90,1] + 70.353;
   1:  PR[GP1:91,2] = PR[GP1:90,2] + -12.026;
   1:L PR[91] 10mm/sec CNT100;
   1:  PR[GP1:91,1] = PR[GP1:90,1] + 72.635;
   1:  PR[GP1:91,2] = PR[GP1:90,2] + 0.277;
   1:L PR[91] 10mm/sec CNT100;
   1:  PR[GP1:91,1] = PR[GP1:90,1] + 72.311;
   1:  PR[GP1:91,2] = PR[GP1:90,2] + 1.966;
   1:L PR[91] 10mm/sec CNT100;
   1:  PR[GP1:91,1] = PR[GP1:90,1] + 70.353;
   1:  PR[GP1:91,2] = PR[GP1:90,2] + 12.584;
   1:L PR[91] 10mm/sec CNT100;
   1:  PR[GP1:91,1] = PR[GP1:90,1] + 63.844;
   1:  PR[GP1:91,2] = PR[GP1:90,2] + 23.258;
   1:L PR[91] 10mm/sec CNT100;
   1:  PR[GP1:91,1] = PR[GP1:90,1] + 53.960;
   1:  PR[GP1:91,2] = PR[GP1:90,2] + 30.940;
   1:L PR[91] 10mm/sec CNT100;
   1:  PR[GP1:91,1] = PR[GP1:90,1] + 52.755;
   1:  PR[GP1:91,2] = PR[GP1:90,2] + 31.376;
   1:L PR[91] 10mm/sec CNT100;
   1:  PR[GP1:91,1] = PR[GP1:90,1] + 42.091;
   1:  PR[GP1:91,2] = PR[GP1:90,2] + 34.760;
   1:L PR[91] 10mm/sec CNT100;
   1:  PR[GP1:91,1] = PR[GP1:90,1] + 37.931;
   1:  PR[GP1:91,2] = PR[GP1:90,2] + 34.793;
   1:L PR[91] 10mm/sec CNT100;
   1:  PR[GP1:91,1] = PR[GP1:90,1] + 29.804;
   1:  PR[GP1:91,2] = PR[GP1:90,2] + 34.441;
   1:L PR[91] 10mm/sec CNT100;
   1:  PR[GP1:91,1] = PR[GP1:90,1] + 22.640;
   1:  PR[GP1:91,2] = PR[GP1:90,2] + 31.978;
   1:L PR[91] 10mm/sec CNT100;
   1:  PR[GP1:91,1] = PR[GP1:90,1] + 18.520;
   1:  PR[GP1:91,2] = PR[GP1:90,2] + 30.259;
   1:L PR[91] 10mm/sec CNT100;
   1:  PR[GP1:91,1] = PR[GP1:90,1] + 10.066;
   1:  PR[GP1:91,2] = PR[GP1:90,2] + 23.495;
   1:L PR[91] 10mm/sec CNT100;
   1:  PR[GP1:91,1] = PR[GP1:90,1] + 9.365;
   1:  PR[GP1:91,2] = PR[GP1:90,2] + 22.834;
   1:L PR[91] 10mm/sec CNT100;
   1:  PR[GP1:91,1] = PR[GP1:90,1] + 6.637;
   1:  PR[GP1:91,2] = PR[GP1:90,2] + 18.334;
   1:L PR[91] 10mm/sec CNT100;
   1:  PR[GP1:91,1] = PR[GP1:90,1] + 3.447;
   1:  PR[GP1:91,2] = PR[GP1:90,2] + 13.251;
   1:L PR[91] 10mm/sec CNT100;
   1:  PR[GP1:91,1] = PR[GP1:90,1] + 2.884;
   1:  PR[GP1:91,2] = PR[GP1:90,2] + 12.466;
   1:L PR[91] 10mm/sec CNT100;
   1:  PR[GP1:91,1] = PR[GP1:90,1] + -3.439;
   1:L PR[91] 10mm/sec CNT100;
   1:  PR[GP1:91,1] = PR[GP1:90,1] + -7.166;
   1:  PR[GP1:91,2] = PR[GP1:90,2] + 18.336;
   1:L PR[91] 10mm/sec CNT100;
   1:  PR[GP1:91,1] = PR[GP1:90,1] + -9.897;
   1:  PR[GP1:91,2] = PR[GP1:90,2] + 22.849;
   1:L PR[91] 10mm/sec CNT100;
   1:  PR[GP1:91,1] = PR[GP1:90,1] + -10.599;
   1:  PR[GP1:91,2] = PR[GP1:90,2] + 23.509;
   1:L PR[91] 10mm/sec CNT100;
   1:  PR[GP1:91,1] = PR[GP1:90,1] + -19.055;
   1:  PR[GP1:91,2] = PR[GP1:90,2] + 30.261;
   1:L PR[91] 10mm/sec CNT100;
   1:  PR[GP1:91,1] = PR[GP1:90,1] + -23.177;
   1:  PR[GP1:91,2] = PR[GP1:90,2] + 31.980;
   1:L PR[91] 10mm/sec CNT100;
   1:  PR[GP1:91,1] = PR[GP1:90,1] + -30.340;
   1:  PR[GP1:91,2] = PR[GP1:90,2] + 34.444;
   1:L PR[91] 10mm/sec CNT100;
   1:  PR[GP1:91,1] = PR[GP1:90,1] + -38.468;
   1:  PR[GP1:91,2] = PR[GP1:90,2] + 34.792;
   1:L PR[91] 10mm/sec CNT100;
   1:  PR[GP1:91,1] = PR[GP1:90,1] + -42.626;
   1:  PR[GP1:91,2] = PR[GP1:90,2] + 34.758;
   1:L PR[91] 10mm/sec CNT100;
   1:  PR[GP1:91,1] = PR[GP1:90,1] + -53.289;
   1:  PR[GP1:91,2] = PR[GP1:90,2] + 31.372;
   1:L PR[91] 10mm/sec CNT100;
   1:  PR[GP1:91,1] = PR[GP1:90,1] + -54.493;
   1:  PR[GP1:91,2] = PR[GP1:90,2] + 30.936;
   1:L PR[91] 10mm/sec CNT100;
   1:  PR[GP1:91,1] = PR[GP1:90,1] + -64.373;
   1:  PR[GP1:91,2] = PR[GP1:90,2] + 23.258;
   1:L PR[91] 10mm/sec CNT100;
   1:  PR[GP1:91,1] = PR[GP1:90,1] + -70.881;
   1:  PR[GP1:91,2] = PR[GP1:90,2] + 12.572;
   1:L PR[91] 10mm/sec CNT100;
   1:  PR[GP1:91,1] = PR[GP1:90,1] + -73.161;
   1:  PR[GP1:91,2] = PR[GP1:90,2] + 0.281;
   1:L PR[91] 10mm/sec CNT100;
   1:  PR[GP1:91,1] = PR[GP1:90,1] + -72.837;
   1:  PR[GP1:91,2] = PR[GP1:90,2] + -1.407;
   1:L PR[91] 10mm/sec CNT100;
   1:  PR[GP1:91,1] = PR[GP1:90,1] + -70.880;
   1:  PR[GP1:91,2] = PR[GP1:90,2] + -12.014;
   1:L PR[91] 10mm/sec CNT100;
   1:  PR[GP1:91,1] = PR[GP1:90,1] + -64.373;
   1:  PR[GP1:91,2] = PR[GP1:90,2] + -22.700;
   1:L PR[91] 10mm/sec CNT100;
   1:  PR[GP1:91,1] = PR[GP1:90,1] + -61.280;
   1:  PR[GP1:91,2] = PR[GP1:90,2] + -25.106;
   1:L PR[91] 10mm/sec CNT100;
   1:  PR[GP1:91,1] = PR[GP1:90,1] + -54.493;
   1:  PR[GP1:91,2] = PR[GP1:90,2] + -30.378;
   1:L PR[91] 10mm/sec CNT100;
   1:  PR[GP1:91,1] = PR[GP1:90,1] + -53.289;
   1:  PR[GP1:91,2] = PR[GP1:90,2] + -30.814;
   1:L PR[91] 10mm/sec CNT100;
   1:  PR[GP1:91,1] = PR[GP1:90,1] + -42.626;
   1:  PR[GP1:91,2] = PR[GP1:90,2] + -34.200;
   1:L PR[91] 10mm/sec CNT100;
   1:  PR[GP1:91,1] = PR[GP1:90,1] + -38.468;
   1:  PR[GP1:91,2] = PR[GP1:90,2] + -34.234;
   1:L PR[91] 10mm/sec CNT100;
   1:  PR[GP1:91,1] = PR[GP1:90,1] + -30.340;
   1:  PR[GP1:91,2] = PR[GP1:90,2] + -33.886;
   1:L PR[91] 10mm/sec CNT100;
   1:  PR[GP1:91,1] = PR[GP1:90,1] + -23.177;
   1:  PR[GP1:91,2] = PR[GP1:90,2] + -31.422;
   1:L PR[91] 10mm/sec CNT100;
   1:  PR[GP1:91,1] = PR[GP1:90,1] + -19.055;
   1:  PR[GP1:91,2] = PR[GP1:90,2] + -29.703;
   1:L PR[91] 10mm/sec CNT100;
   1:  PR[GP1:91,1] = PR[GP1:90,1] + -10.599;
   1:  PR[GP1:91,2] = PR[GP1:90,2] + -22.951;
   1:L PR[91] 10mm/sec CNT100;
   1:  PR[GP1:91,1] = PR[GP1:90,1] + -9.897;
   1:  PR[GP1:91,2] = PR[GP1:90,2] + -22.291;
   1:L PR[91] 10mm/sec CNT100;
   1:  PR[GP1:91,1] = PR[GP1:90,1] + -7.164;
   1:  PR[GP1:91,2] = PR[GP1:90,2] + -17.775;
   1:L PR[91] 10mm/sec CNT100;
   1:  PR[GP1:91,1] = PR[GP1:90,1] + -3.977;
   1:  PR[GP1:91,2] = PR[GP1:90,2] + -12.690;
   1:L PR[91] 10mm/sec CNT100;
   1:  PR[GP1:91,1] = PR[GP1:90,1] + -3.417;
   1:  PR[GP1:91,2] = PR[GP1:90,2] + -11.908;
   1:L PR[91] 10mm/sec CNT100;
   1:  PR[GP1:91,1] = PR[GP1:90,1] + 2.905;
   1:L PR[91] 10mm/sec CNT100;
   1:  PR[GP1:91,1] = PR[GP1:90,1] + 9.309;
   1:  PR[GP1:91,2] = PR[GP1:90,2] + -22.465;
   1:  PR[GP1:91,3] = PR[GP1:90,3] + 30.805;
   1:L PR[91] 10mm/sec CNT100;
   1:  PR[GP1:91,1] = PR[GP1:90,1] + 18.538;
   1:  PR[GP1:91,2] = PR[GP1:90,2] + -29.840;
   1:L PR[91] 10mm/sec CNT100;
   1:  PR[GP1:91,1] = PR[GP1:90,1] + 21.614;
   1:  PR[GP1:91,2] = PR[GP1:90,2] + -31.124;
   1:L PR[91] 10mm/sec CNT100;
   1:  PR[GP1:91,1] = PR[GP1:90,1] + 29.814;
   1:  PR[GP1:91,2] = PR[GP1:90,2] + -33.943;
   1:L PR[91] 10mm/sec CNT100;
   1:  PR[GP1:91,1] = PR[GP1:90,1] + 36.897;
   1:  PR[GP1:91,2] = PR[GP1:90,2] + -34.250;
   1:L PR[91] 10mm/sec CNT100;
   1:  PR[GP1:91,1] = PR[GP1:90,1] + 42.072;
   1:  PR[GP1:91,2] = PR[GP1:90,2] + -34.209;
   1:L PR[91] 10mm/sec CNT100;
   1:  PR[GP1:91,1] = PR[GP1:90,1] + 51.836;
   1:  PR[GP1:91,2] = PR[GP1:90,2] + -31.111;
   1:L PR[91] 10mm/sec CNT100;
   1:  PR[GP1:91,1] = PR[GP1:90,1] + 53.906;
   1:  PR[GP1:91,2] = PR[GP1:90,2] + -30.362;
   1:L PR[91] 10mm/sec CNT100;
   1:  PR[GP1:91,1] = PR[GP1:90,1] + 63.683;
   1:  PR[GP1:91,2] = PR[GP1:90,2] + -22.766;
   1:L PR[91] 10mm/sec CNT100;
   1:  PR[GP1:91,1] = PR[GP1:90,1] + 63.788;
   1:  PR[GP1:91,2] = PR[GP1:90,2] + -22.679;
   1:L PR[91] 10mm/sec CNT100;
   1:  PR[GP1:91,1] = PR[GP1:90,1] + 70.296;
   1:  PR[GP1:91,2] = PR[GP1:90,2] + -12.007;
   1:L PR[91] 10mm/sec CNT100;
   1:  PR[GP1:91,1] = PR[GP1:90,1] + 72.569;
   1:  PR[GP1:91,2] = PR[GP1:90,2] + 0.279;
   1:L PR[91] 10mm/sec CNT100;
   1:  PR[GP1:91,1] = PR[GP1:90,1] + 70.295;
   1:  PR[GP1:91,2] = PR[GP1:90,2] + 12.565;
   1:L PR[91] 10mm/sec CNT100;
   1:  PR[GP1:91,1] = PR[GP1:90,1] + 63.788;
   1:  PR[GP1:91,2] = PR[GP1:90,2] + 23.237;
   1:L PR[91] 10mm/sec CNT100;
   1:  PR[GP1:91,1] = PR[GP1:90,1] + 63.683;
   1:  PR[GP1:91,2] = PR[GP1:90,2] + 23.324;
   1:L PR[91] 10mm/sec CNT100;
   1:  PR[GP1:91,1] = PR[GP1:90,1] + 53.906;
   1:  PR[GP1:91,2] = PR[GP1:90,2] + 30.920;
   1:L PR[91] 10mm/sec CNT100;
   1:  PR[GP1:91,1] = PR[GP1:90,1] + 51.836;
   1:  PR[GP1:91,2] = PR[GP1:90,2] + 31.669;
   1:L PR[91] 10mm/sec CNT100;
   1:  PR[GP1:91,1] = PR[GP1:90,1] + 42.072;
   1:  PR[GP1:91,2] = PR[GP1:90,2] + 34.767;
   1:L PR[91] 10mm/sec CNT100;
   1:  PR[GP1:91,1] = PR[GP1:90,1] + 36.897;
   1:  PR[GP1:91,2] = PR[GP1:90,2] + 34.808;
   1:L PR[91] 10mm/sec CNT100;
   1:  PR[GP1:91,1] = PR[GP1:90,1] + 29.814;
   1:  PR[GP1:91,2] = PR[GP1:90,2] + 34.501;
   1:L PR[91] 10mm/sec CNT100;
   1:  PR[GP1:91,1] = PR[GP1:90,1] + 21.614;
   1:  PR[GP1:91,2] = PR[GP1:90,2] + 31.682;
   1:L PR[91] 10mm/sec CNT100;
   1:  PR[GP1:91,1] = PR[GP1:90,1] + 18.538;
   1:  PR[GP1:91,2] = PR[GP1:90,2] + 30.398;
   1:L PR[91] 10mm/sec CNT100;
   1:  PR[GP1:91,1] = PR[GP1:90,1] + 9.311;
   1:  PR[GP1:91,2] = PR[GP1:90,2] + 23.025;
   1:L PR[91] 10mm/sec CNT100;
   1:  PR[GP1:91,1] = PR[GP1:90,1] + 3.672;
   1:  PR[GP1:91,2] = PR[GP1:90,2] + 14.038;
   1:L PR[91] 10mm/sec CNT100;
   1:  PR[GP1:91,1] = PR[GP1:90,1] + 2.777;
   1:  PR[GP1:91,2] = PR[GP1:90,2] + 12.791;
   1:L PR[91] 10mm/sec CNT100;
   1:  PR[GP1:91,1] = PR[GP1:90,1] + -3.331;
   1:L PR[91] 10mm/sec CNT100;
   1:  PR[GP1:91,1] = PR[GP1:90,1] + -9.841;
   1:  PR[GP1:91,2] = PR[GP1:90,2] + 23.037;
   1:L PR[91] 10mm/sec CNT100;
   1:  PR[GP1:91,1] = PR[GP1:90,1] + -19.072;
   1:  PR[GP1:91,2] = PR[GP1:90,2] + 30.400;
   1:L PR[91] 10mm/sec CNT100;
   1:  PR[GP1:91,1] = PR[GP1:90,1] + -22.150;
   1:  PR[GP1:91,2] = PR[GP1:90,2] + 31.684;
   1:L PR[91] 10mm/sec CNT100;
   1:  PR[GP1:91,1] = PR[GP1:90,1] + -30.349;
   1:  PR[GP1:91,2] = PR[GP1:90,2] + 34.504;
   1:L PR[91] 10mm/sec CNT100;
   1:  PR[GP1:91,1] = PR[GP1:90,1] + -37.433;
   1:  PR[GP1:91,2] = PR[GP1:90,2] + 34.807;
   1:L PR[91] 10mm/sec CNT100;
   1:  PR[GP1:91,1] = PR[GP1:90,1] + -42.607;
   1:  PR[GP1:91,2] = PR[GP1:90,2] + 34.765;
   1:L PR[91] 10mm/sec CNT100;
   1:  PR[GP1:91,1] = PR[GP1:90,1] + -52.370;
   1:  PR[GP1:91,2] = PR[GP1:90,2] + 31.664;
   1:L PR[91] 10mm/sec CNT100;
   1:  PR[GP1:91,1] = PR[GP1:90,1] + -54.438;
   1:  PR[GP1:91,2] = PR[GP1:90,2] + 30.915;
   1:L PR[91] 10mm/sec CNT100;
   1:  PR[GP1:91,1] = PR[GP1:90,1] + -64.213;
   1:  PR[GP1:91,2] = PR[GP1:90,2] + 23.323;
   1:L PR[91] 10mm/sec CNT100;
   1:  PR[GP1:91,1] = PR[GP1:90,1] + -64.318;
   1:  PR[GP1:91,2] = PR[GP1:90,2] + 23.237;
   1:L PR[91] 10mm/sec CNT100;
   1:  PR[GP1:91,1] = PR[GP1:90,1] + -70.823;
   1:  PR[GP1:91,2] = PR[GP1:90,2] + 12.553;
   1:L PR[91] 10mm/sec CNT100;
   1:  PR[GP1:91,1] = PR[GP1:90,1] + -73.095;
   1:  PR[GP1:91,2] = PR[GP1:90,2] + 0.279;
   1:L PR[91] 10mm/sec CNT100;
   1:  PR[GP1:91,1] = PR[GP1:90,1] + -70.823;
   1:  PR[GP1:91,2] = PR[GP1:90,2] + -11.995;
   1:L PR[91] 10mm/sec CNT100;
   1:  PR[GP1:91,1] = PR[GP1:90,1] + -65.634;
   1:  PR[GP1:91,2] = PR[GP1:90,2] + -20.529;
   1:L PR[91] 10mm/sec CNT100;
   1:  PR[GP1:91,1] = PR[GP1:90,1] + -64.323;
   1:  PR[GP1:91,2] = PR[GP1:90,2] + -22.671;
   1:L PR[91] 10mm/sec CNT100;
   1:  PR[GP1:91,1] = PR[GP1:90,1] + -54.438;
   1:  PR[GP1:91,2] = PR[GP1:90,2] + -30.357;
   1:L PR[91] 10mm/sec CNT100;
   1:  PR[GP1:91,1] = PR[GP1:90,1] + -52.369;
   1:  PR[GP1:91,2] = PR[GP1:90,2] + -31.106;
   1:L PR[91] 10mm/sec CNT100;
   1:  PR[GP1:91,1] = PR[GP1:90,1] + -42.607;
   1:  PR[GP1:91,2] = PR[GP1:90,2] + -34.207;
   1:L PR[91] 10mm/sec CNT100;
   1:  PR[GP1:91,1] = PR[GP1:90,1] + -37.433;
   1:  PR[GP1:91,2] = PR[GP1:90,2] + -34.249;
   1:L PR[91] 10mm/sec CNT100;
   1:  PR[GP1:91,1] = PR[GP1:90,1] + -30.349;
   1:  PR[GP1:91,2] = PR[GP1:90,2] + -33.946;
   1:L PR[91] 10mm/sec CNT100;
   1:  PR[GP1:91,1] = PR[GP1:90,1] + -22.150;
   1:  PR[GP1:91,2] = PR[GP1:90,2] + -31.126;
   1:L PR[91] 10mm/sec CNT100;
   1:  PR[GP1:91,1] = PR[GP1:90,1] + -19.072;
   1:  PR[GP1:91,2] = PR[GP1:90,2] + -29.841;
   1:L PR[91] 10mm/sec CNT100;
   1:  PR[GP1:91,1] = PR[GP1:90,1] + -9.843;
   1:  PR[GP1:91,2] = PR[GP1:90,2] + -22.480;
   1:L PR[91] 10mm/sec CNT100;
   1:  PR[GP1:91,1] = PR[GP1:90,1] + -4.199;
   1:  PR[GP1:91,2] = PR[GP1:90,2] + -13.476;
   1:L PR[91] 10mm/sec CNT100;
   1:  PR[GP1:91,1] = PR[GP1:90,1] + -3.309;
   1:  PR[GP1:91,2] = PR[GP1:90,2] + -12.233;
   1:L PR[91] 10mm/sec CNT100;
   1:  PR[GP1:91,1] = PR[GP1:90,1] + 2.798;
   1:L PR[91] 10mm/sec CNT100;
   1:  PR[GP1:91,1] = PR[GP1:90,1] + 8.538;
   1:  PR[GP1:91,2] = PR[GP1:90,2] + -21.752;
   1:  PR[GP1:91,3] = PR[GP1:90,3] + 31.415;
   1:L PR[91] 10mm/sec CNT100;
   1:  PR[GP1:91,1] = PR[GP1:90,1] + 9.040;
   1:  PR[GP1:91,2] = PR[GP1:90,2] + -22.471;
   1:L PR[91] 10mm/sec CNT100;
   1:  PR[GP1:91,1] = PR[GP1:90,1] + 9.451;
   1:  PR[GP1:91,2] = PR[GP1:90,2] + -22.841;
   1:L PR[91] 10mm/sec CNT100;
   1:  PR[GP1:91,1] = PR[GP1:90,1] + 12.538;
   1:  PR[GP1:91,2] = PR[GP1:90,2] + -25.165;
   1:L PR[91] 10mm/sec CNT100;
   1:  PR[GP1:91,1] = PR[GP1:90,1] + 18.556;
   1:  PR[GP1:91,2] = PR[GP1:90,2] + -29.980;
   1:L PR[91] 10mm/sec CNT100;
   1:  PR[GP1:91,1] = PR[GP1:90,1] + 20.588;
   1:  PR[GP1:91,2] = PR[GP1:90,2] + -30.827;
   1:L PR[91] 10mm/sec CNT100;
   1:  PR[GP1:91,1] = PR[GP1:90,1] + 29.824;
   1:  PR[GP1:91,2] = PR[GP1:90,2] + -34.003;
   1:L PR[91] 10mm/sec CNT100;
   1:  PR[GP1:91,1] = PR[GP1:90,1] + 35.862;
   1:  PR[GP1:91,2] = PR[GP1:90,2] + -34.265;
   1:L PR[91] 10mm/sec CNT100;
   1:  PR[GP1:91,1] = PR[GP1:90,1] + 42.053;
   1:  PR[GP1:91,2] = PR[GP1:90,2] + -34.215;
   1:L PR[91] 10mm/sec CNT100;
   1:  PR[GP1:91,1] = PR[GP1:90,1] + 50.916;
   1:  PR[GP1:91,2] = PR[GP1:90,2] + -31.403;
   1:L PR[91] 10mm/sec CNT100;
   1:  PR[GP1:91,1] = PR[GP1:90,1] + 53.851;
   1:  PR[GP1:91,2] = PR[GP1:90,2] + -30.341;
   1:L PR[91] 10mm/sec CNT100;
   1:  PR[GP1:91,1] = PR[GP1:90,1] + 62.961;
   1:  PR[GP1:91,2] = PR[GP1:90,2] + -23.264;
   1:L PR[91] 10mm/sec CNT100;
   1:  PR[GP1:91,1] = PR[GP1:90,1] + 63.702;
   1:  PR[GP1:91,2] = PR[GP1:90,2] + -22.652;
   1:L PR[91] 10mm/sec CNT100;
   1:  PR[GP1:91,1] = PR[GP1:90,1] + 70.238;
   1:  PR[GP1:91,2] = PR[GP1:90,2] + -11.987;
   1:L PR[91] 10mm/sec CNT100;
   1:  PR[GP1:91,1] = PR[GP1:90,1] + 72.503;
   1:  PR[GP1:91,2] = PR[GP1:90,2] + 0.279;
   1:L PR[91] 10mm/sec CNT100;
   1:  PR[GP1:91,1] = PR[GP1:90,1] + 70.238;
   1:  PR[GP1:91,2] = PR[GP1:90,2] + 12.545;
   1:L PR[91] 10mm/sec CNT100;
   1:  PR[GP1:91,1] = PR[GP1:90,1] + 63.702;
   1:  PR[GP1:91,2] = PR[GP1:90,2] + 23.210;
   1:L PR[91] 10mm/sec CNT100;
   1:  PR[GP1:91,1] = PR[GP1:90,1] + 62.961;
   1:  PR[GP1:91,2] = PR[GP1:90,2] + 23.822;
   1:L PR[91] 10mm/sec CNT100;
   1:  PR[GP1:91,1] = PR[GP1:90,1] + 53.851;
   1:  PR[GP1:91,2] = PR[GP1:90,2] + 30.900;
   1:L PR[91] 10mm/sec CNT100;
   1:  PR[GP1:91,1] = PR[GP1:90,1] + 50.916;
   1:  PR[GP1:91,2] = PR[GP1:90,2] + 31.961;
   1:L PR[91] 10mm/sec CNT100;
   1:  PR[GP1:91,1] = PR[GP1:90,1] + 42.053;
   1:  PR[GP1:91,2] = PR[GP1:90,2] + 34.773;
   1:L PR[91] 10mm/sec CNT100;
   1:  PR[GP1:91,1] = PR[GP1:90,1] + 35.862;
   1:  PR[GP1:91,2] = PR[GP1:90,2] + 34.823;
   1:L PR[91] 10mm/sec CNT100;
   1:  PR[GP1:91,1] = PR[GP1:90,1] + 29.825;
   1:  PR[GP1:91,2] = PR[GP1:90,2] + 34.561;
   1:L PR[91] 10mm/sec CNT100;
   1:  PR[GP1:91,1] = PR[GP1:90,1] + 20.588;
   1:  PR[GP1:91,2] = PR[GP1:90,2] + 31.385;
   1:L PR[91] 10mm/sec CNT100;
   1:  PR[GP1:91,1] = PR[GP1:90,1] + 18.556;
   1:  PR[GP1:91,2] = PR[GP1:90,2] + 30.538;
   1:L PR[91] 10mm/sec CNT100;
   1:  PR[GP1:91,1] = PR[GP1:90,1] + 12.538;
   1:  PR[GP1:91,2] = PR[GP1:90,2] + 25.723;
   1:L PR[91] 10mm/sec CNT100;
   1:  PR[GP1:91,1] = PR[GP1:90,1] + 9.452;
   1:  PR[GP1:91,2] = PR[GP1:90,2] + 23.400;
   1:L PR[91] 10mm/sec CNT100;
   1:  PR[GP1:91,1] = PR[GP1:90,1] + 9.051;
   1:  PR[GP1:91,2] = PR[GP1:90,2] + 23.039;
   1:L PR[91] 10mm/sec CNT100;
   1:  PR[GP1:91,1] = PR[GP1:90,1] + 3.897;
   1:  PR[GP1:91,2] = PR[GP1:90,2] + 14.825;
   1:L PR[91] 10mm/sec CNT100;
   1:  PR[GP1:91,1] = PR[GP1:90,1] + 2.670;
   1:  PR[GP1:91,2] = PR[GP1:90,2] + 13.116;
   1:L PR[91] 10mm/sec CNT100;
   1:  PR[GP1:91,1] = PR[GP1:90,1] + -3.223;
   1:L PR[91] 10mm/sec CNT100;
   1:  PR[GP1:91,1] = PR[GP1:90,1] + -9.070;
   1:  PR[GP1:91,2] = PR[GP1:90,2] + 22.324;
   1:L PR[91] 10mm/sec CNT100;
   1:  PR[GP1:91,1] = PR[GP1:90,1] + -9.567;
   1:  PR[GP1:91,2] = PR[GP1:90,2] + 23.038;
   1:L PR[91] 10mm/sec CNT100;
   1:  PR[GP1:91,1] = PR[GP1:90,1] + -9.980;
   1:  PR[GP1:91,2] = PR[GP1:90,2] + 23.410;
   1:L PR[91] 10mm/sec CNT100;
   1:  PR[GP1:91,1] = PR[GP1:90,1] + -13.064;
   1:  PR[GP1:91,2] = PR[GP1:90,2] + 25.728;
   1:L PR[91] 10mm/sec CNT100;
   1:  PR[GP1:91,1] = PR[GP1:90,1] + -19.089;
   1:  PR[GP1:91,2] = PR[GP1:90,2] + 30.538;
   1:L PR[91] 10mm/sec CNT100;
   1:  PR[GP1:91,1] = PR[GP1:90,1] + -21.123;
   1:  PR[GP1:91,2] = PR[GP1:90,2] + 31.387;
   1:L PR[91] 10mm/sec CNT100;
   1:  PR[GP1:91,1] = PR[GP1:90,1] + -30.359;
   1:  PR[GP1:91,2] = PR[GP1:90,2] + 34.563;
   1:L PR[91] 10mm/sec CNT100;
   1:  PR[GP1:91,1] = PR[GP1:90,1] + -36.398;
   1:  PR[GP1:91,2] = PR[GP1:90,2] + 34.822;
   1:L PR[91] 10mm/sec CNT100;
   1:  PR[GP1:91,1] = PR[GP1:90,1] + -42.588;
   1:  PR[GP1:91,2] = PR[GP1:90,2] + 34.772;
   1:L PR[91] 10mm/sec CNT100;
   1:  PR[GP1:91,1] = PR[GP1:90,1] + -51.450;
   1:  PR[GP1:91,2] = PR[GP1:90,2] + 31.957;
   1:L PR[91] 10mm/sec CNT100;
   1:  PR[GP1:91,1] = PR[GP1:90,1] + -54.383;
   1:  PR[GP1:91,2] = PR[GP1:90,2] + 30.895;
   1:L PR[91] 10mm/sec CNT100;
   1:  PR[GP1:91,1] = PR[GP1:90,1] + -63.492;
   1:  PR[GP1:91,2] = PR[GP1:90,2] + 23.821;
   1:L PR[91] 10mm/sec CNT100;
   1:  PR[GP1:91,1] = PR[GP1:90,1] + -64.232;
   1:  PR[GP1:91,2] = PR[GP1:90,2] + 23.211;
   1:L PR[91] 10mm/sec CNT100;
   1:  PR[GP1:91,1] = PR[GP1:90,1] + -70.765;
   1:  PR[GP1:91,2] = PR[GP1:90,2] + 12.532;
   1:L PR[91] 10mm/sec CNT100;
   1:  PR[GP1:91,1] = PR[GP1:90,1] + -73.029;
   1:  PR[GP1:91,2] = PR[GP1:90,2] + 0.279;
   1:L PR[91] 10mm/sec CNT100;
   1:  PR[GP1:91,1] = PR[GP1:90,1] + -70.765;
   1:  PR[GP1:91,2] = PR[GP1:90,2] + -11.975;
   1:L PR[91] 10mm/sec CNT100;
   1:  PR[GP1:91,1] = PR[GP1:90,1] + -70.136;
   1:  PR[GP1:91,2] = PR[GP1:90,2] + -13.009;
   1:L PR[91] 10mm/sec CNT100;
   1:  PR[GP1:91,1] = PR[GP1:90,1] + -64.232;
   1:  PR[GP1:91,2] = PR[GP1:90,2] + -22.652;
   1:L PR[91] 10mm/sec CNT100;
   1:  PR[GP1:91,1] = PR[GP1:90,1] + -63.492;
   1:  PR[GP1:91,2] = PR[GP1:90,2] + -23.263;
   1:L PR[91] 10mm/sec CNT100;
   1:  PR[GP1:91,1] = PR[GP1:90,1] + -54.383;
   1:  PR[GP1:91,2] = PR[GP1:90,2] + -30.337;
   1:L PR[91] 10mm/sec CNT100;
   1:  PR[GP1:91,1] = PR[GP1:90,1] + -51.450;
   1:  PR[GP1:91,2] = PR[GP1:90,2] + -31.399;
   1:L PR[91] 10mm/sec CNT100;
   1:  PR[GP1:91,1] = PR[GP1:90,1] + -42.588;
   1:  PR[GP1:91,2] = PR[GP1:90,2] + -34.214;
   1:L PR[91] 10mm/sec CNT100;
   1:  PR[GP1:91,1] = PR[GP1:90,1] + -36.398;
   1:  PR[GP1:91,2] = PR[GP1:90,2] + -34.264;
   1:L PR[91] 10mm/sec CNT100;
   1:  PR[GP1:91,1] = PR[GP1:90,1] + -30.359;
   1:  PR[GP1:91,2] = PR[GP1:90,2] + -34.005;
   1:L PR[91] 10mm/sec CNT100;
   1:  PR[GP1:91,1] = PR[GP1:90,1] + -21.123;
   1:  PR[GP1:91,2] = PR[GP1:90,2] + -30.829;
   1:L PR[91] 10mm/sec CNT100;
   1:  PR[GP1:91,1] = PR[GP1:90,1] + -19.089;
   1:  PR[GP1:91,2] = PR[GP1:90,2] + -29.980;
   1:L PR[91] 10mm/sec CNT100;
   1:  PR[GP1:91,1] = PR[GP1:90,1] + -13.064;
   1:  PR[GP1:91,2] = PR[GP1:90,2] + -25.170;
   1:L PR[91] 10mm/sec CNT100;
   1:  PR[GP1:91,1] = PR[GP1:90,1] + -9.980;
   1:  PR[GP1:91,2] = PR[GP1:90,2] + -22.852;
   1:L PR[91] 10mm/sec CNT100;
   1:  PR[GP1:91,1] = PR[GP1:90,1] + -9.578;
   1:  PR[GP1:91,2] = PR[GP1:90,2] + -22.490;
   1:L PR[91] 10mm/sec CNT100;
   1:  PR[GP1:91,1] = PR[GP1:90,1] + -4.420;
   1:  PR[GP1:91,2] = PR[GP1:90,2] + -14.261;
   1:L PR[91] 10mm/sec CNT100;
   1:  PR[GP1:91,1] = PR[GP1:90,1] + -3.202;
   1:  PR[GP1:91,2] = PR[GP1:90,2] + -12.558;
   1:L PR[91] 10mm/sec CNT100;
   1:  PR[GP1:91,1] = PR[GP1:90,1] + 2.692;
   1:L PR[91] 10mm/sec CNT100;
   1:  PR[GP1:91,1] = PR[GP1:90,1] + 7.768;
   1:  PR[GP1:91,2] = PR[GP1:90,2] + -21.034;
   1:  PR[GP1:91,3] = PR[GP1:90,3] + 32.025;
   1:L PR[91] 10mm/sec CNT100;
   1:  PR[GP1:91,1] = PR[GP1:90,1] + 8.770;
   1:  PR[GP1:91,2] = PR[GP1:90,2] + -22.469;
   1:L PR[91] 10mm/sec CNT100;
   1:  PR[GP1:91,1] = PR[GP1:90,1] + 9.622;
   1:  PR[GP1:91,2] = PR[GP1:90,2] + -23.237;
   1:L PR[91] 10mm/sec CNT100;
   1:  PR[GP1:91,1] = PR[GP1:90,1] + 15.537;
   1:  PR[GP1:91,2] = PR[GP1:90,2] + -27.690;
   1:L PR[91] 10mm/sec CNT100;
   1:  PR[GP1:91,1] = PR[GP1:90,1] + 18.573;
   1:  PR[GP1:91,2] = PR[GP1:90,2] + -30.119;
   1:L PR[91] 10mm/sec CNT100;
   1:  PR[GP1:91,1] = PR[GP1:90,1] + 19.561;
   1:  PR[GP1:91,2] = PR[GP1:90,2] + -30.531;
   1:L PR[91] 10mm/sec CNT100;
   1:  PR[GP1:91,1] = PR[GP1:90,1] + 29.835;
   1:  PR[GP1:91,2] = PR[GP1:90,2] + -34.064;
   1:L PR[91] 10mm/sec CNT100;
   1:  PR[GP1:91,1] = PR[GP1:90,1] + 34.827;
   1:  PR[GP1:91,2] = PR[GP1:90,2] + -34.280;
   1:L PR[91] 10mm/sec CNT100;
   1:  PR[GP1:91,1] = PR[GP1:90,1] + 42.035;
   1:  PR[GP1:91,2] = PR[GP1:90,2] + -34.222;
   1:L PR[91] 10mm/sec CNT100;
   1:  PR[GP1:91,1] = PR[GP1:90,1] + 49.997;
   1:  PR[GP1:91,2] = PR[GP1:90,2] + -31.696;
   1:L PR[91] 10mm/sec CNT100;
   1:  PR[GP1:91,1] = PR[GP1:90,1] + 53.797;
   1:  PR[GP1:91,2] = PR[GP1:90,2] + -30.321;
   1:L PR[91] 10mm/sec CNT100;
   1:  PR[GP1:91,1] = PR[GP1:90,1] + 62.239;
   1:  PR[GP1:91,2] = PR[GP1:90,2] + -23.762;
   1:L PR[91] 10mm/sec CNT100;
   1:  PR[GP1:91,1] = PR[GP1:90,1] + 63.615;
   1:  PR[GP1:91,2] = PR[GP1:90,2] + -22.626;
   1:L PR[91] 10mm/sec CNT100;
   1:  PR[GP1:91,1] = PR[GP1:90,1] + 69.873;
   1:  PR[GP1:91,2] = PR[GP1:90,2] + -12.421;
   1:L PR[91] 10mm/sec CNT100;
   1:  PR[GP1:91,1] = PR[GP1:90,1] + 70.136;
   1:  PR[GP1:91,2] = PR[GP1:90,2] + -11.975;
   1:L PR[91] 10mm/sec CNT100;
   1:  PR[GP1:91,1] = PR[GP1:90,1] + 72.429;
   1:  PR[GP1:91,2] = PR[GP1:90,2] + 0.279;
   1:L PR[91] 10mm/sec CNT100;
   1:  PR[GP1:91,1] = PR[GP1:90,1] + 70.995;
   1:  PR[GP1:91,2] = PR[GP1:90,2] + 7.998;
   1:L PR[91] 10mm/sec CNT100;
   1:  PR[GP1:91,1] = PR[GP1:90,1] + 70.137;
   1:  PR[GP1:91,2] = PR[GP1:90,2] + 12.532;
   1:L PR[91] 10mm/sec CNT100;
   1:  PR[GP1:91,1] = PR[GP1:90,1] + 69.873;
   1:  PR[GP1:91,2] = PR[GP1:90,2] + 12.980;
   1:L PR[91] 10mm/sec CNT100;
   1:  PR[GP1:91,1] = PR[GP1:90,1] + 63.615;
   1:  PR[GP1:91,2] = PR[GP1:90,2] + 23.184;
   1:L PR[91] 10mm/sec CNT100;
   1:  PR[GP1:91,1] = PR[GP1:90,1] + 62.239;
   1:  PR[GP1:91,2] = PR[GP1:90,2] + 24.320;
   1:L PR[91] 10mm/sec CNT100;
   1:  PR[GP1:91,1] = PR[GP1:90,1] + 53.797;
   1:  PR[GP1:91,2] = PR[GP1:90,2] + 30.879;
   1:L PR[91] 10mm/sec CNT100;
   1:  PR[GP1:91,1] = PR[GP1:90,1] + 49.997;
   1:  PR[GP1:91,2] = PR[GP1:90,2] + 32.254;
   1:L PR[91] 10mm/sec CNT100;
   1:  PR[GP1:91,1] = PR[GP1:90,1] + 42.035;
   1:  PR[GP1:91,2] = PR[GP1:90,2] + 34.780;
   1:L PR[91] 10mm/sec CNT100;
   1:  PR[GP1:91,1] = PR[GP1:90,1] + 34.827;
   1:  PR[GP1:91,2] = PR[GP1:90,2] + 34.838;
   1:L PR[91] 10mm/sec CNT100;
   1:  PR[GP1:91,1] = PR[GP1:90,1] + 29.835;
   1:  PR[GP1:91,2] = PR[GP1:90,2] + 34.622;
   1:L PR[91] 10mm/sec CNT100;
   1:  PR[GP1:91,1] = PR[GP1:90,1] + 19.562;
   1:  PR[GP1:91,2] = PR[GP1:90,2] + 31.089;
   1:L PR[91] 10mm/sec CNT100;
   1:  PR[GP1:91,1] = PR[GP1:90,1] + 18.574;
   1:  PR[GP1:91,2] = PR[GP1:90,2] + 30.677;
   1:L PR[91] 10mm/sec CNT100;
   1:  PR[GP1:91,1] = PR[GP1:90,1] + 15.537;
   1:  PR[GP1:91,2] = PR[GP1:90,2] + 28.248;
   1:L PR[91] 10mm/sec CNT100;
   1:  PR[GP1:91,1] = PR[GP1:90,1] + 9.622;
   1:  PR[GP1:91,2] = PR[GP1:90,2] + 23.795;
   1:L PR[91] 10mm/sec CNT100;
   1:  PR[GP1:91,1] = PR[GP1:90,1] + 8.781;
   1:  PR[GP1:91,2] = PR[GP1:90,2] + 23.037;
   1:L PR[91] 10mm/sec CNT100;
   1:  PR[GP1:91,1] = PR[GP1:90,1] + 4.122;
   1:  PR[GP1:91,2] = PR[GP1:90,2] + 15.613;
   1:L PR[91] 10mm/sec CNT100;
   1:  PR[GP1:91,1] = PR[GP1:90,1] + 2.563;
   1:  PR[GP1:91,2] = PR[GP1:90,2] + 13.441;
   1:L PR[91] 10mm/sec CNT100;
   1:  PR[GP1:91,1] = PR[GP1:90,1] + -3.115;
   1:L PR[91] 10mm/sec CNT100;
   1:  PR[GP1:91,1] = PR[GP1:90,1] + -8.299;
   1:  PR[GP1:91,2] = PR[GP1:90,2] + 21.604;
   1:L PR[91] 10mm/sec CNT100;
   1:  PR[GP1:91,1] = PR[GP1:90,1] + -9.292;
   1:  PR[GP1:91,2] = PR[GP1:90,2] + 23.032;
   1:L PR[91] 10mm/sec CNT100;
   1:  PR[GP1:91,1] = PR[GP1:90,1] + -10.148;
   1:  PR[GP1:91,2] = PR[GP1:90,2] + 23.803;
   1:L PR[91] 10mm/sec CNT100;
   1:  PR[GP1:91,1] = PR[GP1:90,1] + -16.063;
   1:  PR[GP1:91,2] = PR[GP1:90,2] + 28.248;
   1:L PR[91] 10mm/sec CNT100;
   1:  PR[GP1:91,1] = PR[GP1:90,1] + -19.106;
   1:  PR[GP1:91,2] = PR[GP1:90,2] + 30.677;
   1:L PR[91] 10mm/sec CNT100;
   1:  PR[GP1:91,1] = PR[GP1:90,1] + -20.097;
   1:  PR[GP1:91,2] = PR[GP1:90,2] + 31.090;
   1:L PR[91] 10mm/sec CNT100;
   1:  PR[GP1:91,1] = PR[GP1:90,1] + -30.369;
   1:  PR[GP1:91,2] = PR[GP1:90,2] + 34.623;
   1:L PR[91] 10mm/sec CNT100;
   1:  PR[GP1:91,1] = PR[GP1:90,1] + -35.362;
   1:  PR[GP1:91,2] = PR[GP1:90,2] + 34.837;
   1:L PR[91] 10mm/sec CNT100;
   1:  PR[GP1:91,1] = PR[GP1:90,1] + -42.569;
   1:  PR[GP1:91,2] = PR[GP1:90,2] + 34.779;
   1:L PR[91] 10mm/sec CNT100;
   1:  PR[GP1:91,1] = PR[GP1:90,1] + -50.531;
   1:  PR[GP1:91,2] = PR[GP1:90,2] + 32.250;
   1:L PR[91] 10mm/sec CNT100;
   1:  PR[GP1:91,1] = PR[GP1:90,1] + -54.329;
   1:  PR[GP1:91,2] = PR[GP1:90,2] + 30.875;
   1:L PR[91] 10mm/sec CNT100;
   1:  PR[GP1:91,1] = PR[GP1:90,1] + -62.770;
   1:  PR[GP1:91,2] = PR[GP1:90,2] + 24.319;
   1:L PR[91] 10mm/sec CNT100;
   1:  PR[GP1:91,1] = PR[GP1:90,1] + -64.145;
   1:  PR[GP1:91,2] = PR[GP1:90,2] + 23.185;
   1:L PR[91] 10mm/sec CNT100;
   1:  PR[GP1:91,1] = PR[GP1:90,1] + -70.400;
   1:  PR[GP1:91,2] = PR[GP1:90,2] + 12.968;
   1:L PR[91] 10mm/sec CNT100;
   1:  PR[GP1:91,1] = PR[GP1:90,1] + -70.663;
   1:  PR[GP1:91,2] = PR[GP1:90,2] + 12.520;
   1:L PR[91] 10mm/sec CNT100;
   1:  PR[GP1:91,1] = PR[GP1:90,1] + -72.955;
   1:  PR[GP1:91,2] = PR[GP1:90,2] + 0.279;
   1:L PR[91] 10mm/sec CNT100;
   1:  PR[GP1:91,1] = PR[GP1:90,1] + -71.521;
   1:  PR[GP1:91,2] = PR[GP1:90,2] + -7.434;
   1:L PR[91] 10mm/sec CNT100;
   1:  PR[GP1:91,1] = PR[GP1:90,1] + -70.664;
   1:  PR[GP1:91,2] = PR[GP1:90,2] + -11.961;
   1:L PR[91] 10mm/sec CNT100;
   1:  PR[GP1:91,1] = PR[GP1:90,1] + -70.400;
   1:  PR[GP1:91,2] = PR[GP1:90,2] + -12.410;
   1:L PR[91] 10mm/sec CNT100;
   1:  PR[GP1:91,1] = PR[GP1:90,1] + -64.145;
   1:  PR[GP1:91,2] = PR[GP1:90,2] + -22.627;
   1:L PR[91] 10mm/sec CNT100;
   1:  PR[GP1:91,1] = PR[GP1:90,1] + -62.770;
   1:  PR[GP1:91,2] = PR[GP1:90,2] + -23.760;
   1:L PR[91] 10mm/sec CNT100;
   1:  PR[GP1:91,1] = PR[GP1:90,1] + -54.329;
   1:  PR[GP1:91,2] = PR[GP1:90,2] + -30.317;
   1:L PR[91] 10mm/sec CNT100;
   1:  PR[GP1:91,1] = PR[GP1:90,1] + -50.531;
   1:  PR[GP1:91,2] = PR[GP1:90,2] + -31.692;
   1:L PR[91] 10mm/sec CNT100;
   1:  PR[GP1:91,1] = PR[GP1:90,1] + -42.569;
   1:  PR[GP1:91,2] = PR[GP1:90,2] + -34.221;
   1:L PR[91] 10mm/sec CNT100;
   1:  PR[GP1:91,1] = PR[GP1:90,1] + -35.362;
   1:  PR[GP1:91,2] = PR[GP1:90,2] + -34.279;
   1:L PR[91] 10mm/sec CNT100;
   1:  PR[GP1:91,1] = PR[GP1:90,1] + -30.369;
   1:  PR[GP1:91,2] = PR[GP1:90,2] + -34.065;
   1:L PR[91] 10mm/sec CNT100;
   1:  PR[GP1:91,1] = PR[GP1:90,1] + -20.097;
   1:  PR[GP1:91,2] = PR[GP1:90,2] + -30.532;
   1:L PR[91] 10mm/sec CNT100;
   1:  PR[GP1:91,1] = PR[GP1:90,1] + -19.106;
   1:  PR[GP1:91,2] = PR[GP1:90,2] + -30.119;
   1:L PR[91] 10mm/sec CNT100;
   1:  PR[GP1:91,1] = PR[GP1:90,1] + -16.063;
   1:  PR[GP1:91,2] = PR[GP1:90,2] + -27.690;
   1:L PR[91] 10mm/sec CNT100;
   1:  PR[GP1:91,1] = PR[GP1:90,1] + -10.148;
   1:  PR[GP1:91,2] = PR[GP1:90,2] + -23.245;
   1:L PR[91] 10mm/sec CNT100;
   1:  PR[GP1:91,1] = PR[GP1:90,1] + -9.303;
   1:  PR[GP1:91,2] = PR[GP1:90,2] + -22.484;
   1:L PR[91] 10mm/sec CNT100;
   1:  PR[GP1:91,1] = PR[GP1:90,1] + -4.642;
   1:  PR[GP1:91,2] = PR[GP1:90,2] + -15.046;
   1:L PR[91] 10mm/sec CNT100;
   1:  PR[GP1:91,1] = PR[GP1:90,1] + -3.094;
   1:  PR[GP1:91,2] = PR[GP1:90,2] + -12.883;
   1:L PR[91] 10mm/sec CNT100;
   1:  PR[GP1:91,1] = PR[GP1:90,1] + 2.585;
   1:L PR[91] 10mm/sec CNT100;
   1:  PR[GP1:91,1] = PR[GP1:90,1] + 6.998;
   1:  PR[GP1:91,2] = PR[GP1:90,2] + -20.316;
   1:  PR[GP1:91,3] = PR[GP1:90,3] + 32.635;
   1:L PR[91] 10mm/sec CNT100;
   1:  PR[GP1:91,1] = PR[GP1:90,1] + 8.500;
   1:  PR[GP1:91,2] = PR[GP1:90,2] + -22.468;
   1:L PR[91] 10mm/sec CNT100;
   1:  PR[GP1:91,1] = PR[GP1:90,1] + 9.792;
   1:  PR[GP1:91,2] = PR[GP1:90,2] + -23.632;
   1:L PR[91] 10mm/sec CNT100;
   1:  PR[GP1:91,1] = PR[GP1:90,1] + 18.567;
   1:  PR[GP1:91,2] = PR[GP1:90,2] + -30.243;
   1:L PR[91] 10mm/sec CNT100;
   1:  PR[GP1:91,1] = PR[GP1:90,1] + 29.845;
   1:  PR[GP1:91,2] = PR[GP1:90,2] + -34.124;
   1:L PR[91] 10mm/sec CNT100;
   1:  PR[GP1:91,1] = PR[GP1:90,1] + 33.792;
   1:  PR[GP1:91,2] = PR[GP1:90,2] + -34.294;
   1:L PR[91] 10mm/sec CNT100;
   1:  PR[GP1:91,1] = PR[GP1:90,1] + 42.016;
   1:  PR[GP1:91,2] = PR[GP1:90,2] + -34.229;
   1:L PR[91] 10mm/sec CNT100;
   1:  PR[GP1:91,1] = PR[GP1:90,1] + 49.078;
   1:  PR[GP1:91,2] = PR[GP1:90,2] + -31.988;
   1:L PR[91] 10mm/sec CNT100;
   1:  PR[GP1:91,1] = PR[GP1:90,1] + 53.742;
   1:  PR[GP1:91,2] = PR[GP1:90,2] + -30.301;
   1:L PR[91] 10mm/sec CNT100;
   1:  PR[GP1:91,1] = PR[GP1:90,1] + 61.517;
   1:  PR[GP1:91,2] = PR[GP1:90,2] + -24.261;
   1:L PR[91] 10mm/sec CNT100;
   1:  PR[GP1:91,1] = PR[GP1:90,1] + 63.529;
   1:  PR[GP1:91,2] = PR[GP1:90,2] + -22.600;
   1:L PR[91] 10mm/sec CNT100;
   1:  PR[GP1:91,1] = PR[GP1:90,1] + 69.389;
   1:  PR[GP1:91,2] = PR[GP1:90,2] + -13.044;
   1:L PR[91] 10mm/sec CNT100;
   1:  PR[GP1:91,1] = PR[GP1:90,1] + 70.028;
   1:  PR[GP1:91,2] = PR[GP1:90,2] + -11.959;
   1:L PR[91] 10mm/sec CNT100;
   1:  PR[GP1:91,1] = PR[GP1:90,1] + 72.177;
   1:  PR[GP1:91,2] = PR[GP1:90,2] + -0.447;
   1:L PR[91] 10mm/sec CNT100;
   1:  PR[GP1:91,1] = PR[GP1:90,1] + 72.335;
   1:  PR[GP1:91,2] = PR[GP1:90,2] + 0.287;
   1:L PR[91] 10mm/sec CNT100;
   1:  PR[GP1:91,1] = PR[GP1:90,1] + 70.210;
   1:  PR[GP1:91,2] = PR[GP1:90,2] + 11.488;
   1:L PR[91] 10mm/sec CNT100;
   1:  PR[GP1:91,1] = PR[GP1:90,1] + 70.026;
   1:  PR[GP1:91,2] = PR[GP1:90,2] + 12.519;
   1:L PR[91] 10mm/sec CNT100;
   1:  PR[GP1:91,1] = PR[GP1:90,1] + 69.389;
   1:  PR[GP1:91,2] = PR[GP1:90,2] + 13.602;
   1:L PR[91] 10mm/sec CNT100;
   1:  PR[GP1:91,1] = PR[GP1:90,1] + 63.529;
   1:  PR[GP1:91,2] = PR[GP1:90,2] + 23.158;
   1:L PR[91] 10mm/sec CNT100;
   1:  PR[GP1:91,1] = PR[GP1:90,1] + 61.517;
   1:  PR[GP1:91,2] = PR[GP1:90,2] + 24.818;
   1:L PR[91] 10mm/sec CNT100;
   1:  PR[GP1:91,1] = PR[GP1:90,1] + 53.742;
   1:  PR[GP1:91,2] = PR[GP1:90,2] + 30.859;
   1:L PR[91] 10mm/sec CNT100;
   1:  PR[GP1:91,1] = PR[GP1:90,1] + 49.078;
   1:  PR[GP1:91,2] = PR[GP1:90,2] + 32.546;
   1:L PR[91] 10mm/sec CNT100;
   1:  PR[GP1:91,1] = PR[GP1:90,1] + 42.016;
   1:  PR[GP1:91,2] = PR[GP1:90,2] + 34.787;
   1:L PR[91] 10mm/sec CNT100;
   1:  PR[GP1:91,1] = PR[GP1:90,1] + 33.792;
   1:  PR[GP1:91,2] = PR[GP1:90,2] + 34.853;
   1:L PR[91] 10mm/sec CNT100;
   1:  PR[GP1:91,1] = PR[GP1:90,1] + 29.845;
   1:  PR[GP1:91,2] = PR[GP1:90,2] + 34.682;
   1:L PR[91] 10mm/sec CNT100;
   1:  PR[GP1:91,1] = PR[GP1:90,1] + 18.575;
   1:  PR[GP1:91,2] = PR[GP1:90,2] + 30.806;
   1:L PR[91] 10mm/sec CNT100;
   1:  PR[GP1:91,1] = PR[GP1:90,1] + 9.792;
   1:  PR[GP1:91,2] = PR[GP1:90,2] + 24.190;
   1:L PR[91] 10mm/sec CNT100;
   1:  PR[GP1:91,1] = PR[GP1:90,1] + 8.511;
   1:  PR[GP1:91,2] = PR[GP1:90,2] + 23.036;
   1:L PR[91] 10mm/sec CNT100;
   1:  PR[GP1:91,1] = PR[GP1:90,1] + 4.347;
   1:  PR[GP1:91,2] = PR[GP1:90,2] + 16.400;
   1:L PR[91] 10mm/sec CNT100;
   1:  PR[GP1:91,1] = PR[GP1:90,1] + 2.456;
   1:  PR[GP1:91,2] = PR[GP1:90,2] + 13.766;
   1:L PR[91] 10mm/sec CNT100;
   1:  PR[GP1:91,1] = PR[GP1:90,1] + -3.007;
   1:L PR[91] 10mm/sec CNT100;
   1:  PR[GP1:91,1] = PR[GP1:90,1] + -7.528;
   1:  PR[GP1:91,2] = PR[GP1:90,2] + 20.885;
   1:L PR[91] 10mm/sec CNT100;
   1:  PR[GP1:91,1] = PR[GP1:90,1] + -9.018;
   1:  PR[GP1:91,2] = PR[GP1:90,2] + 23.025;
   1:L PR[91] 10mm/sec CNT100;
   1:  PR[GP1:91,1] = PR[GP1:90,1] + -10.316;
   1:  PR[GP1:91,2] = PR[GP1:90,2] + 24.195;
   1:L PR[91] 10mm/sec CNT100;
   1:  PR[GP1:91,1] = PR[GP1:90,1] + -19.099;
   1:  PR[GP1:91,2] = PR[GP1:90,2] + 30.801;
   1:L PR[91] 10mm/sec CNT100;
   1:  PR[GP1:91,1] = PR[GP1:90,1] + -30.379;
   1:  PR[GP1:91,2] = PR[GP1:90,2] + 34.683;
   1:L PR[91] 10mm/sec CNT100;
   1:  PR[GP1:91,1] = PR[GP1:90,1] + -34.327;
   1:  PR[GP1:91,2] = PR[GP1:90,2] + 34.853;
   1:L PR[91] 10mm/sec CNT100;
   1:  PR[GP1:91,1] = PR[GP1:90,1] + -42.550;
   1:  PR[GP1:91,2] = PR[GP1:90,2] + 34.786;
   1:L PR[91] 10mm/sec CNT100;
   1:  PR[GP1:91,1] = PR[GP1:90,1] + -49.611;
   1:  PR[GP1:91,2] = PR[GP1:90,2] + 32.543;
   1:L PR[91] 10mm/sec CNT100;
   1:  PR[GP1:91,1] = PR[GP1:90,1] + -54.274;
   1:  PR[GP1:91,2] = PR[GP1:90,2] + 30.854;
   1:L PR[91] 10mm/sec CNT100;
   1:  PR[GP1:91,1] = PR[GP1:90,1] + -62.048;
   1:  PR[GP1:91,2] = PR[GP1:90,2] + 24.816;
   1:L PR[91] 10mm/sec CNT100;
   1:  PR[GP1:91,1] = PR[GP1:90,1] + -64.058;
   1:  PR[GP1:91,2] = PR[GP1:90,2] + 23.159;
   1:L PR[91] 10mm/sec CNT100;
   1:  PR[GP1:91,1] = PR[GP1:90,1] + -69.916;
   1:  PR[GP1:91,2] = PR[GP1:90,2] + 13.591;
   1:L PR[91] 10mm/sec CNT100;
   1:  PR[GP1:91,1] = PR[GP1:90,1] + -70.555;
   1:  PR[GP1:91,2] = PR[GP1:90,2] + 12.503;
   1:L PR[91] 10mm/sec CNT100;
   1:  PR[GP1:91,1] = PR[GP1:90,1] + -72.703;
   1:  PR[GP1:91,2] = PR[GP1:90,2] + 1.004;
   1:L PR[91] 10mm/sec CNT100;
   1:  PR[GP1:91,1] = PR[GP1:90,1] + -72.861;
   1:  PR[GP1:91,2] = PR[GP1:90,2] + 0.270;
   1:L PR[91] 10mm/sec CNT100;
   1:  PR[GP1:91,1] = PR[GP1:90,1] + -72.446;
   1:  PR[GP1:91,2] = PR[GP1:90,2] + -1.962;
   1:L PR[91] 10mm/sec CNT100;
   1:  PR[GP1:91,1] = PR[GP1:90,1] + -70.737;
   1:  PR[GP1:91,2] = PR[GP1:90,2] + -10.918;
   1:L PR[91] 10mm/sec CNT100;
   1:  PR[GP1:91,1] = PR[GP1:90,1] + -70.553;
   1:  PR[GP1:91,2] = PR[GP1:90,2] + -11.947;
   1:L PR[91] 10mm/sec CNT100;
   1:  PR[GP1:91,1] = PR[GP1:90,1] + -69.916;
   1:  PR[GP1:91,2] = PR[GP1:90,2] + -13.033;
   1:L PR[91] 10mm/sec CNT100;
   1:  PR[GP1:91,1] = PR[GP1:90,1] + -64.058;
   1:  PR[GP1:91,2] = PR[GP1:90,2] + -22.601;
   1:L PR[91] 10mm/sec CNT100;
   1:  PR[GP1:91,1] = PR[GP1:90,1] + -62.048;
   1:  PR[GP1:91,2] = PR[GP1:90,2] + -24.258;
   1:L PR[91] 10mm/sec CNT100;
   1:  PR[GP1:91,1] = PR[GP1:90,1] + -54.274;
   1:  PR[GP1:91,2] = PR[GP1:90,2] + -30.296;
   1:L PR[91] 10mm/sec CNT100;
   1:  PR[GP1:91,1] = PR[GP1:90,1] + -49.611;
   1:  PR[GP1:91,2] = PR[GP1:90,2] + -31.985;
   1:L PR[91] 10mm/sec CNT100;
   1:  PR[GP1:91,1] = PR[GP1:90,1] + -42.550;
   1:  PR[GP1:91,2] = PR[GP1:90,2] + -34.228;
   1:L PR[91] 10mm/sec CNT100;
   1:  PR[GP1:91,1] = PR[GP1:90,1] + -34.327;
   1:  PR[GP1:91,2] = PR[GP1:90,2] + -34.294;
   1:L PR[91] 10mm/sec CNT100;
   1:  PR[GP1:91,1] = PR[GP1:90,1] + -30.379;
   1:  PR[GP1:91,2] = PR[GP1:90,2] + -34.125;
   1:L PR[91] 10mm/sec CNT100;
   1:  PR[GP1:91,1] = PR[GP1:90,1] + -19.100;
   1:  PR[GP1:91,2] = PR[GP1:90,2] + -30.243;
   1:L PR[91] 10mm/sec CNT100;
   1:  PR[GP1:91,1] = PR[GP1:90,1] + -10.316;
   1:  PR[GP1:91,2] = PR[GP1:90,2] + -23.637;
   1:L PR[91] 10mm/sec CNT100;
   1:  PR[GP1:91,1] = PR[GP1:90,1] + -9.029;
   1:  PR[GP1:91,2] = PR[GP1:90,2] + -22.477;
   1:L PR[91] 10mm/sec CNT100;
   1:  PR[GP1:91,1] = PR[GP1:90,1] + -4.863;
   1:  PR[GP1:91,2] = PR[GP1:90,2] + -15.831;
   1:L PR[91] 10mm/sec CNT100;
   1:  PR[GP1:91,1] = PR[GP1:90,1] + -2.986;
   1:  PR[GP1:91,2] = PR[GP1:90,2] + -13.208;
   1:L PR[91] 10mm/sec CNT100;
   1:  PR[GP1:91,1] = PR[GP1:90,1] + 2.478;
   1:L PR[91] 10mm/sec CNT100;
   1:  PR[GP1:91,1] = PR[GP1:90,1] + 6.228;
   1:  PR[GP1:91,2] = PR[GP1:90,2] + -19.598;
   1:  PR[GP1:91,3] = PR[GP1:90,3] + 33.245;
   1:L PR[91] 10mm/sec CNT100;
   1:  PR[GP1:91,1] = PR[GP1:90,1] + 8.230;
   1:  PR[GP1:91,2] = PR[GP1:90,2] + -22.467;
   1:L PR[91] 10mm/sec CNT100;
   1:  PR[GP1:91,1] = PR[GP1:90,1] + 9.962;
   1:  PR[GP1:91,2] = PR[GP1:90,2] + -24.027;
   1:L PR[91] 10mm/sec CNT100;
   1:  PR[GP1:91,1] = PR[GP1:90,1] + 17.995;
   1:  PR[GP1:91,2] = PR[GP1:90,2] + -30.074;
   1:L PR[91] 10mm/sec CNT100;
   1:  PR[GP1:91,1] = PR[GP1:90,1] + 18.497;
   1:  PR[GP1:91,2] = PR[GP1:90,2] + -30.359;
   1:L PR[91] 10mm/sec CNT100;
   1:  PR[GP1:91,1] = PR[GP1:90,1] + 21.352;
   1:  PR[GP1:91,2] = PR[GP1:90,2] + -31.260;
   1:L PR[91] 10mm/sec CNT100;
   1:  PR[GP1:91,1] = PR[GP1:90,1] + 29.855;
   1:  PR[GP1:91,2] = PR[GP1:90,2] + -34.184;
   1:L PR[91] 10mm/sec CNT100;
   1:  PR[GP1:91,1] = PR[GP1:90,1] + 32.757;
   1:  PR[GP1:91,2] = PR[GP1:90,2] + -34.309;
   1:L PR[91] 10mm/sec CNT100;
   1:  PR[GP1:91,1] = PR[GP1:90,1] + 41.998;
   1:  PR[GP1:91,2] = PR[GP1:90,2] + -34.236;
   1:L PR[91] 10mm/sec CNT100;
   1:  PR[GP1:91,1] = PR[GP1:90,1] + 48.159;
   1:  PR[GP1:91,2] = PR[GP1:90,2] + -32.281;
   1:L PR[91] 10mm/sec CNT100;
   1:  PR[GP1:91,1] = PR[GP1:90,1] + 53.688;
   1:  PR[GP1:91,2] = PR[GP1:90,2] + -30.281;
   1:L PR[91] 10mm/sec CNT100;
   1:  PR[GP1:91,1] = PR[GP1:90,1] + 60.795;
   1:  PR[GP1:91,2] = PR[GP1:90,2] + -24.759;
   1:L PR[91] 10mm/sec CNT100;
   1:  PR[GP1:91,1] = PR[GP1:90,1] + 63.442;
   1:  PR[GP1:91,2] = PR[GP1:90,2] + -22.574;
   1:L PR[91] 10mm/sec CNT100;
   1:  PR[GP1:91,1] = PR[GP1:90,1] + 68.905;
   1:  PR[GP1:91,2] = PR[GP1:90,2] + -13.665;
   1:L PR[91] 10mm/sec CNT100;
   1:  PR[GP1:91,1] = PR[GP1:90,1] + 69.919;
   1:  PR[GP1:91,2] = PR[GP1:90,2] + -11.942;
   1:L PR[91] 10mm/sec CNT100;
   1:  PR[GP1:91,1] = PR[GP1:90,1] + 71.940;
   1:  PR[GP1:91,2] = PR[GP1:90,2] + -1.117;
   1:L PR[91] 10mm/sec CNT100;
   1:  PR[GP1:91,1] = PR[GP1:90,1] + 72.175;
   1:  PR[GP1:91,2] = PR[GP1:90,2] + -0.026;
   1:L PR[91] 10mm/sec CNT100;
   1:  PR[GP1:91,1] = PR[GP1:90,1] + 72.229;
   1:  PR[GP1:91,2] = PR[GP1:90,2] + 0.276;
   1:L PR[91] 10mm/sec CNT100;
   1:  PR[GP1:91,1] = PR[GP1:90,1] + 70.211;
   1:  PR[GP1:91,2] = PR[GP1:90,2] + 10.859;
   1:L PR[91] 10mm/sec CNT100;
   1:  PR[GP1:91,1] = PR[GP1:90,1] + 69.918;
   1:  PR[GP1:91,2] = PR[GP1:90,2] + 12.502;
   1:L PR[91] 10mm/sec CNT100;
   1:  PR[GP1:91,1] = PR[GP1:90,1] + 68.905;
   1:  PR[GP1:91,2] = PR[GP1:90,2] + 14.224;
   1:L PR[91] 10mm/sec CNT100;
   1:  PR[GP1:91,1] = PR[GP1:90,1] + 63.442;
   1:  PR[GP1:91,2] = PR[GP1:90,2] + 23.132;
   1:L PR[91] 10mm/sec CNT100;
   1:  PR[GP1:91,1] = PR[GP1:90,1] + 60.796;
   1:  PR[GP1:91,2] = PR[GP1:90,2] + 25.317;
   1:L PR[91] 10mm/sec CNT100;
   1:  PR[GP1:91,1] = PR[GP1:90,1] + 53.688;
   1:  PR[GP1:91,2] = PR[GP1:90,2] + 30.839;
   1:L PR[91] 10mm/sec CNT100;
   1:  PR[GP1:91,1] = PR[GP1:90,1] + 48.159;
   1:  PR[GP1:91,2] = PR[GP1:90,2] + 32.839;
   1:L PR[91] 10mm/sec CNT100;
   1:  PR[GP1:91,1] = PR[GP1:90,1] + 41.998;
   1:  PR[GP1:91,2] = PR[GP1:90,2] + 34.794;
   1:L PR[91] 10mm/sec CNT100;
   1:  PR[GP1:91,1] = PR[GP1:90,1] + 32.757;
   1:  PR[GP1:91,2] = PR[GP1:90,2] + 34.867;
   1:L PR[91] 10mm/sec CNT100;
   1:  PR[GP1:91,1] = PR[GP1:90,1] + 29.855;
   1:  PR[GP1:91,2] = PR[GP1:90,2] + 34.742;
   1:L PR[91] 10mm/sec CNT100;
   1:  PR[GP1:91,1] = PR[GP1:90,1] + 21.353;
   1:  PR[GP1:91,2] = PR[GP1:90,2] + 31.818;
   1:L PR[91] 10mm/sec CNT100;
   1:  PR[GP1:91,1] = PR[GP1:90,1] + 18.850;
   1:  PR[GP1:91,2] = PR[GP1:90,2] + 31.016;
   1:L PR[91] 10mm/sec CNT100;
   1:  PR[GP1:91,1] = PR[GP1:90,1] + 18.491;
   1:  PR[GP1:91,2] = PR[GP1:90,2] + 30.913;
   1:L PR[91] 10mm/sec CNT100;
   1:  PR[GP1:91,1] = PR[GP1:90,1] + 17.995;
   1:  PR[GP1:91,2] = PR[GP1:90,2] + 30.632;
   1:L PR[91] 10mm/sec CNT100;
   1:  PR[GP1:91,1] = PR[GP1:90,1] + 9.962;
